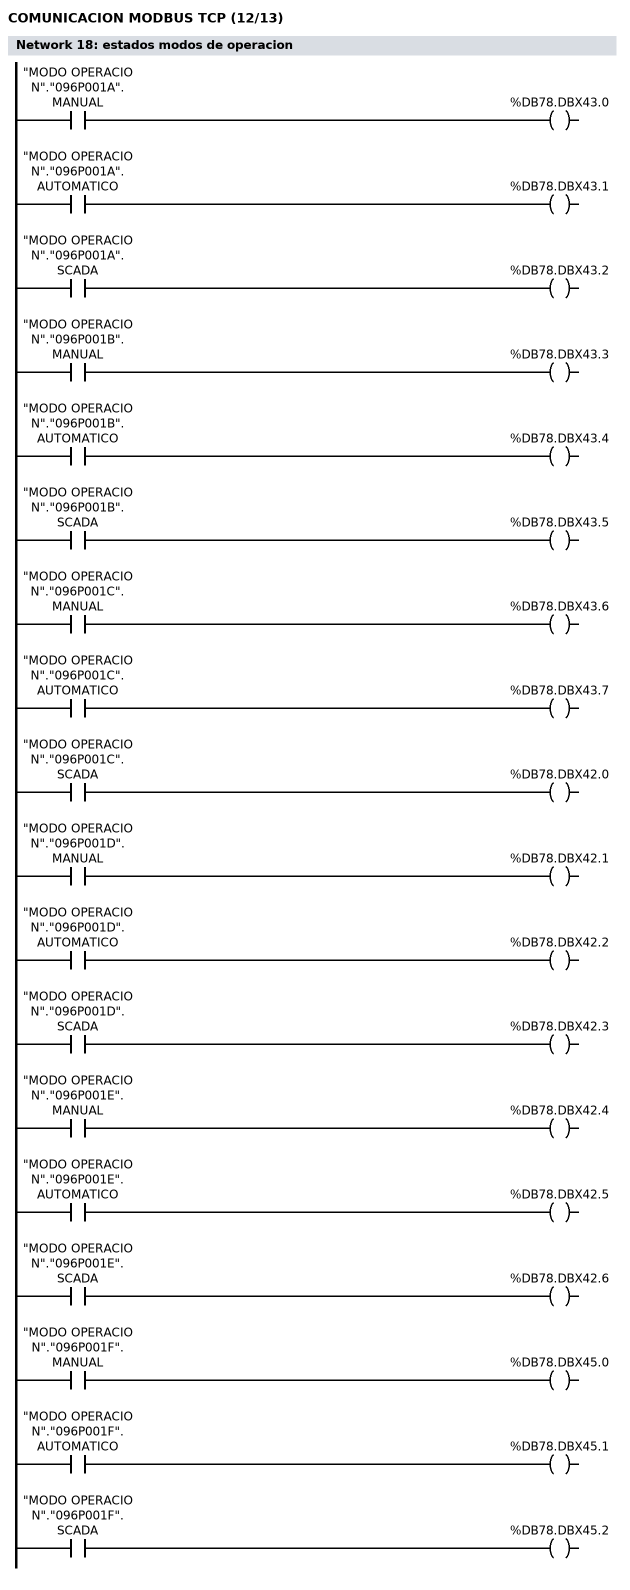
   RUNG wire#powerrail
      Contact( "MODO OPERACION"."096P001A".MANUAL )
      Coil( %DB78.DBX43.0 )
   END_RUNG
   RUNG wire#powerrail
      Contact( "MODO OPERACION"."096P001A".AUTOMATICO )
      Coil( %DB78.DBX43.1 )
   END_RUNG
   RUNG wire#powerrail
      Contact( "MODO OPERACION"."096P001A".SCADA )
      Coil( %DB78.DBX43.2 )
   END_RUNG
   RUNG wire#powerrail
      Contact( "MODO OPERACION"."096P001B".MANUAL )
      Coil( %DB78.DBX43.3 )
   END_RUNG
   RUNG wire#powerrail
      Contact( "MODO OPERACION"."096P001B".AUTOMATICO )
      Coil( %DB78.DBX43.4 )
   END_RUNG
   RUNG wire#powerrail
      Contact( "MODO OPERACION"."096P001B".SCADA )
      Coil( %DB78.DBX43.5 )
   END_RUNG
   RUNG wire#powerrail
      Contact( "MODO OPERACION"."096P001C".MANUAL )
      Coil( %DB78.DBX43.6 )
   END_RUNG
   RUNG wire#powerrail
      Contact( "MODO OPERACION"."096P001C".AUTOMATICO )
      Coil( %DB78.DBX43.7 )
   END_RUNG
   RUNG wire#powerrail
      Contact( "MODO OPERACION"."096P001C".SCADA )
      Coil( %DB78.DBX42.0 )
   END_RUNG
   RUNG wire#powerrail
      Contact( "MODO OPERACION"."096P001D".MANUAL )
      Coil( %DB78.DBX42.1 )
   END_RUNG
   RUNG wire#powerrail
      Contact( "MODO OPERACION"."096P001D".AUTOMATICO )
      Coil( %DB78.DBX42.2 )
   END_RUNG
   RUNG wire#powerrail
      Contact( "MODO OPERACION"."096P001D".SCADA )
      Coil( %DB78.DBX42.3 )
   END_RUNG
   RUNG wire#powerrail
      Contact( "MODO OPERACION"."096P001E".MANUAL )
      Coil( %DB78.DBX42.4 )
   END_RUNG
   RUNG wire#powerrail
      Contact( "MODO OPERACION"."096P001E".AUTOMATICO )
      Coil( %DB78.DBX42.5 )
   END_RUNG
   RUNG wire#powerrail
      Contact( "MODO OPERACION"."096P001E".SCADA )
      Coil( %DB78.DBX42.6 )
   END_RUNG
   RUNG wire#powerrail
      Contact( "MODO OPERACION"."096P001F".MANUAL )
      Coil( %DB78.DBX45.0 )
   END_RUNG
   RUNG wire#powerrail
      Contact( "MODO OPERACION"."096P001F".AUTOMATICO )
      Coil( %DB78.DBX45.1 )
   END_RUNG
   RUNG wire#powerrail
      Contact( "MODO OPERACION"."096P001F".SCADA )
      Coil( %DB78.DBX45.2 )
   END_RUNG
   // the same network as SCL:
   %DB78.DBX43.0 := "MODO OPERACION"."096P001A".MANUAL;
   %DB78.DBX43.1 := "MODO OPERACION"."096P001A".AUTOMATICO;
   %DB78.DBX43.2 := "MODO OPERACION"."096P001A".SCADA;
   %DB78.DBX43.3 := "MODO OPERACION"."096P001B".MANUAL;
   %DB78.DBX43.4 := "MODO OPERACION"."096P001B".AUTOMATICO;
   %DB78.DBX43.5 := "MODO OPERACION"."096P001B".SCADA;
   %DB78.DBX43.6 := "MODO OPERACION"."096P001C".MANUAL;
   %DB78.DBX43.7 := "MODO OPERACION"."096P001C".AUTOMATICO;
   %DB78.DBX42.0 := "MODO OPERACION"."096P001C".SCADA;
   %DB78.DBX42.1 := "MODO OPERACION"."096P001D".MANUAL;
   %DB78.DBX42.2 := "MODO OPERACION"."096P001D".AUTOMATICO;
   %DB78.DBX42.3 := "MODO OPERACION"."096P001D".SCADA;
   %DB78.DBX42.4 := "MODO OPERACION"."096P001E".MANUAL;
   %DB78.DBX42.5 := "MODO OPERACION"."096P001E".AUTOMATICO;
   %DB78.DBX42.6 := "MODO OPERACION"."096P001E".SCADA;
   %DB78.DBX45.0 := "MODO OPERACION"."096P001F".MANUAL;
   %DB78.DBX45.1 := "MODO OPERACION"."096P001F".AUTOMATICO;
   %DB78.DBX45.2 := "MODO OPERACION"."096P001F".SCADA;
END_REGION

REGION Network 19: fallas gnerales
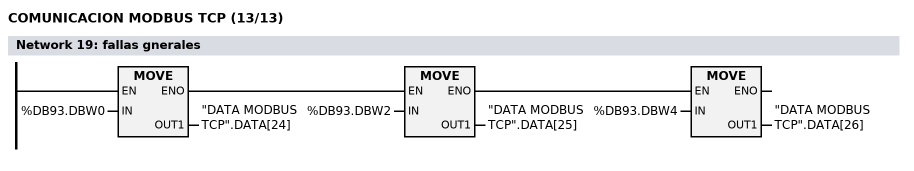
   RUNG wire#powerrail
      Move(in := %DB93.DBW0, out1 => "DATA MODBUS TCP".DATA[24])
      Move(in := %DB93.DBW2, out1 => "DATA MODBUS TCP".DATA[25])
      Move(in := %DB93.DBW4, out1 => "DATA MODBUS TCP".DATA[26])
   END_RUNG
   // the same network as SCL:
   "DATA MODBUS TCP".DATA[24] := %DB93.DBW0;
   "DATA MODBUS TCP".DATA[25] := %DB93.DBW2;
   "DATA MODBUS TCP".DATA[26] := %DB93.DBW4;
END_REGION
END_FUNCTION

FUNCTION "FALLAS" : Void   // FC8, LAD
{ S7_Optimized_Access := 'TRUE' }
VERSION : 0.1
   VAR_TEMP
      "RESET A" : Bool;
      "RESET B" : Bool;
      "RESET C" : Bool;
      "RESET D" : Bool;
      "RESET E" : Bool;
      "RESET F" : Bool;
   END_VAR
BEGIN

REGION Network 1: reset gral
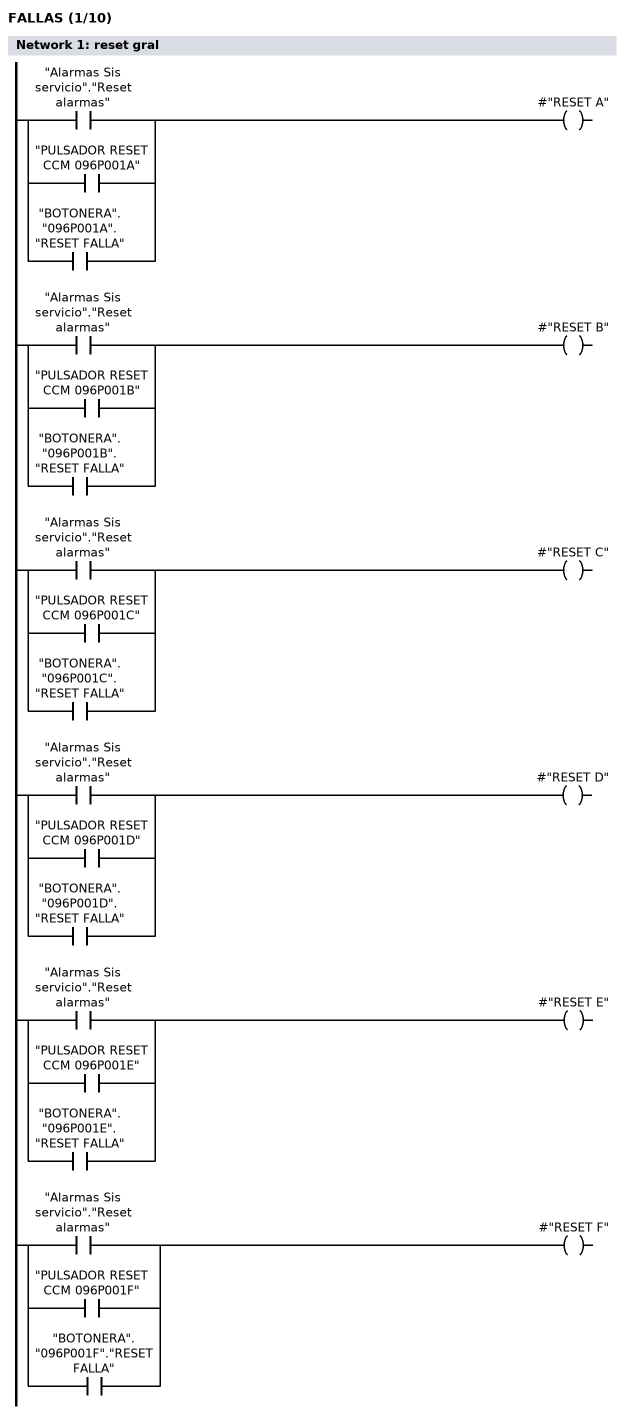
   RUNG wire#powerrail
      Contact( "Alarmas Sis servicio"."Reset alarmas" )
      wire#w1
      Coil( #"RESET A" )
   END_RUNG
   RUNG wire#powerrail
      Contact( "PULSADOR RESET CCM 096P001A" )
   END_RUNG wire#w1
   RUNG wire#powerrail
      Contact( "BOTONERA"."096P001A"."RESET FALLA" )
   END_RUNG wire#w1
   RUNG wire#powerrail
      Contact( "Alarmas Sis servicio"."Reset alarmas" )
      wire#w2
      Coil( #"RESET B" )
   END_RUNG
   RUNG wire#powerrail
      Contact( "PULSADOR RESET CCM 096P001B" )
   END_RUNG wire#w2
   RUNG wire#powerrail
      Contact( "BOTONERA"."096P001B"."RESET FALLA" )
   END_RUNG wire#w2
   RUNG wire#powerrail
      Contact( "Alarmas Sis servicio"."Reset alarmas" )
      wire#w3
      Coil( #"RESET C" )
   END_RUNG
   RUNG wire#powerrail
      Contact( "PULSADOR RESET CCM 096P001C" )
   END_RUNG wire#w3
   RUNG wire#powerrail
      Contact( "BOTONERA"."096P001C"."RESET FALLA" )
   END_RUNG wire#w3
   RUNG wire#powerrail
      Contact( "Alarmas Sis servicio"."Reset alarmas" )
      wire#w4
      Coil( #"RESET D" )
   END_RUNG
   RUNG wire#powerrail
      Contact( "PULSADOR RESET CCM 096P001D" )
   END_RUNG wire#w4
   RUNG wire#powerrail
      Contact( "BOTONERA"."096P001D"."RESET FALLA" )
   END_RUNG wire#w4
   RUNG wire#powerrail
      Contact( "Alarmas Sis servicio"."Reset alarmas" )
      wire#w5
      Coil( #"RESET E" )
   END_RUNG
   RUNG wire#powerrail
      Contact( "PULSADOR RESET CCM 096P001E" )
   END_RUNG wire#w5
   RUNG wire#powerrail
      Contact( "BOTONERA"."096P001E"."RESET FALLA" )
   END_RUNG wire#w5
   RUNG wire#powerrail
      Contact( "Alarmas Sis servicio"."Reset alarmas" )
      wire#w6
      Coil( #"RESET F" )
   END_RUNG
   RUNG wire#powerrail
      Contact( "PULSADOR RESET CCM 096P001F" )
   END_RUNG wire#w6
   RUNG wire#powerrail
      Contact( "BOTONERA"."096P001F"."RESET FALLA" )
   END_RUNG wire#w6
   // the same network as SCL:
   #"RESET A" := "Alarmas Sis servicio"."Reset alarmas" OR "PULSADOR RESET CCM 096P001A" OR "BOTONERA"."096P001A"."RESET FALLA";
   #"RESET B" := "Alarmas Sis servicio"."Reset alarmas" OR "PULSADOR RESET CCM 096P001B" OR "BOTONERA"."096P001B"."RESET FALLA";
   #"RESET C" := "Alarmas Sis servicio"."Reset alarmas" OR "PULSADOR RESET CCM 096P001C" OR "BOTONERA"."096P001C"."RESET FALLA";
   #"RESET D" := "Alarmas Sis servicio"."Reset alarmas" OR "PULSADOR RESET CCM 096P001D" OR "BOTONERA"."096P001D"."RESET FALLA";
   #"RESET E" := "Alarmas Sis servicio"."Reset alarmas" OR "PULSADOR RESET CCM 096P001E" OR "BOTONERA"."096P001E"."RESET FALLA";
   #"RESET F" := "Alarmas Sis servicio"."Reset alarmas" OR "PULSADOR RESET CCM 096P001F" OR "BOTONERA"."096P001F"."RESET FALLA";
END_REGION

REGION Network 2: PARO DE EMERGENCIA GRAL
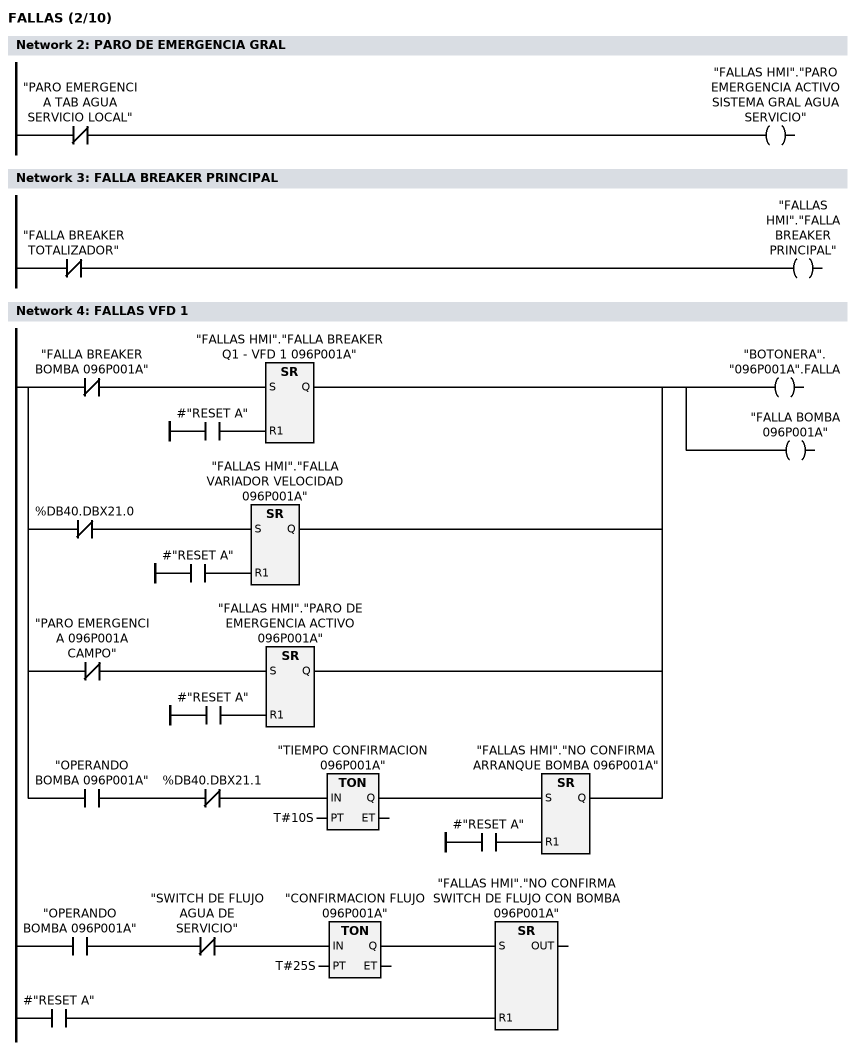
   RUNG wire#powerrail
      I_Contact( "PARO EMERGENCIA TAB AGUA SERVICIO LOCAL" )
      Coil( "FALLAS HMI"."PARO EMERGENCIA ACTIVO SISTEMA GRAL AGUA SERVICIO" )
   END_RUNG
   // the same network as SCL:
   "FALLAS HMI"."PARO EMERGENCIA ACTIVO SISTEMA GRAL AGUA SERVICIO" := NOT "PARO EMERGENCIA TAB AGUA SERVICIO LOCAL";
END_REGION

REGION Network 3: FALLA BREAKER PRINCIPAL
   RUNG wire#powerrail
      I_Contact( "FALLA BREAKER TOTALIZADOR" )
      Coil( "FALLAS HMI"."FALLA BREAKER PRINCIPAL" )
   END_RUNG
   // the same network as SCL:
   "FALLAS HMI"."FALLA BREAKER PRINCIPAL" := NOT "FALLA BREAKER TOTALIZADOR";
END_REGION

REGION Network 4: FALLAS VFD 1
   IF NOT "FALLA BREAKER BOMBA 096P001A" THEN
       "FALLAS HMI"."FALLA BREAKER Q1 - VFD 1 096P001A" := TRUE;   // SR flip-flop
   END_IF;
   IF #"RESET A" THEN "FALLAS HMI"."FALLA BREAKER Q1 - VFD 1 096P001A" := FALSE; END_IF;
   IF NOT %DB40.DBX21.0 THEN
       "FALLAS HMI"."FALLA VARIADOR VELOCIDAD 096P001A" := TRUE;   // SR flip-flop
   END_IF;
   IF #"RESET A" THEN "FALLAS HMI"."FALLA VARIADOR VELOCIDAD 096P001A" := FALSE; END_IF;
   IF NOT "PARO EMERGENCIA 096P001A CAMPO" THEN
       "FALLAS HMI"."PARO DE EMERGENCIA ACTIVO 096P001A" := TRUE;   // SR flip-flop
   END_IF;
   IF #"RESET A" THEN "FALLAS HMI"."PARO DE EMERGENCIA ACTIVO 096P001A" := FALSE; END_IF;
   "TIEMPO CONFIRMACION 096P001A".TON(IN := "OPERANDO BOMBA 096P001A" AND NOT %DB40.DBX21.1, PT := T#10S);
   IF "TIEMPO CONFIRMACION 096P001A".Q THEN
       "FALLAS HMI"."NO CONFIRMA ARRANQUE BOMBA 096P001A" := TRUE;   // SR flip-flop
   END_IF;
   IF #"RESET A" THEN "FALLAS HMI"."NO CONFIRMA ARRANQUE BOMBA 096P001A" := FALSE; END_IF;
   "BOTONERA"."096P001A".FALLA := "FALLAS HMI"."FALLA BREAKER Q1 - VFD 1 096P001A" OR "FALLAS HMI"."FALLA VARIADOR VELOCIDAD 096P001A" OR "FALLAS HMI"."PARO DE EMERGENCIA ACTIVO 096P001A" OR "FALLAS HMI"."NO CONFIRMA ARRANQUE BOMBA 096P001A";
   "FALLA BOMBA 096P001A" := "BOTONERA"."096P001A".FALLA;
   "CONFIRMACION FLUJO 096P001A".TON(IN := "OPERANDO BOMBA 096P001A" AND NOT "SWITCH DE FLUJO AGUA DE SERVICIO",
                           PT := T#25S);
   IF "CONFIRMACION FLUJO 096P001A".Q THEN
       "FALLAS HMI"."NO CONFIRMA SWITCH DE FLUJO CON BOMBA 096P001A" := TRUE;   // SR flip-flop
   END_IF;
   IF #"RESET A" THEN "FALLAS HMI"."NO CONFIRMA SWITCH DE FLUJO CON BOMBA 096P001A" := FALSE; END_IF;
END_REGION

REGION Network 5: FALLAS VFD 2
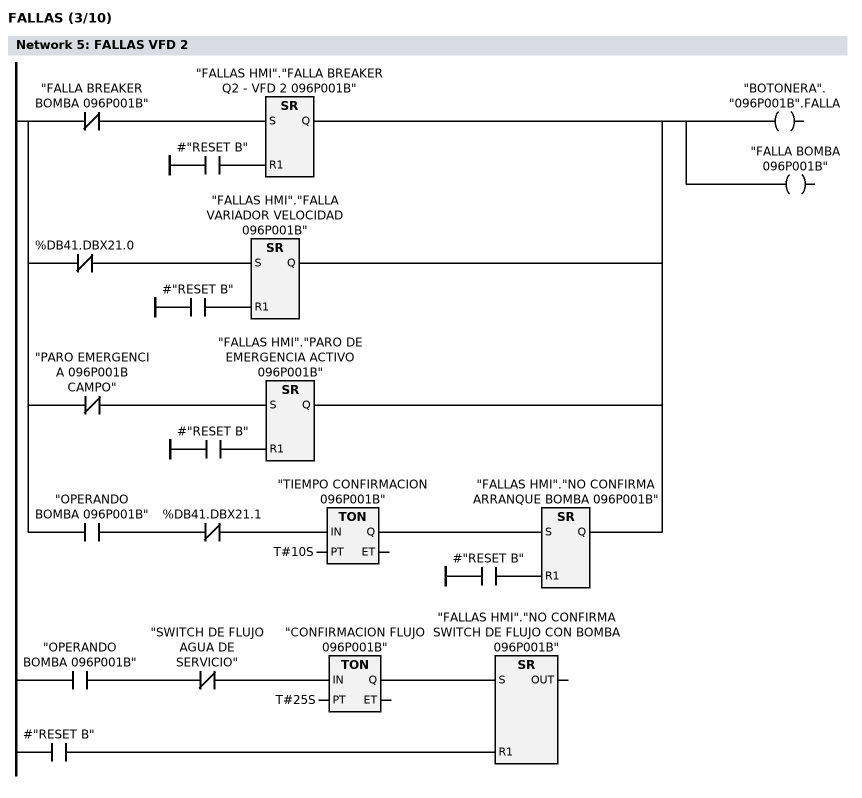
   IF NOT "FALLA BREAKER BOMBA 096P001B" THEN
       "FALLAS HMI"."FALLA BREAKER Q2 - VFD 2 096P001B" := TRUE;   // SR flip-flop
   END_IF;
   IF #"RESET B" THEN "FALLAS HMI"."FALLA BREAKER Q2 - VFD 2 096P001B" := FALSE; END_IF;
   IF NOT %DB41.DBX21.0 THEN
       "FALLAS HMI"."FALLA VARIADOR VELOCIDAD 096P001B" := TRUE;   // SR flip-flop
   END_IF;
   IF #"RESET B" THEN "FALLAS HMI"."FALLA VARIADOR VELOCIDAD 096P001B" := FALSE; END_IF;
   IF NOT "PARO EMERGENCIA 096P001B CAMPO" THEN
       "FALLAS HMI"."PARO DE EMERGENCIA ACTIVO 096P001B" := TRUE;   // SR flip-flop
   END_IF;
   IF #"RESET B" THEN "FALLAS HMI"."PARO DE EMERGENCIA ACTIVO 096P001B" := FALSE; END_IF;
   "TIEMPO CONFIRMACION 096P001B".TON(IN := "OPERANDO BOMBA 096P001B" AND NOT %DB41.DBX21.1, PT := T#10S);
   IF "TIEMPO CONFIRMACION 096P001B".Q THEN
       "FALLAS HMI"."NO CONFIRMA ARRANQUE BOMBA 096P001B" := TRUE;   // SR flip-flop
   END_IF;
   IF #"RESET B" THEN "FALLAS HMI"."NO CONFIRMA ARRANQUE BOMBA 096P001B" := FALSE; END_IF;
   "BOTONERA"."096P001B".FALLA := "FALLAS HMI"."FALLA BREAKER Q2 - VFD 2 096P001B" OR "FALLAS HMI"."FALLA VARIADOR VELOCIDAD 096P001B" OR "FALLAS HMI"."PARO DE EMERGENCIA ACTIVO 096P001B" OR "FALLAS HMI"."NO CONFIRMA ARRANQUE BOMBA 096P001B";
   "FALLA BOMBA 096P001B" := "BOTONERA"."096P001B".FALLA;
   "CONFIRMACION FLUJO 096P001B".TON(IN := "OPERANDO BOMBA 096P001B" AND NOT "SWITCH DE FLUJO AGUA DE SERVICIO",
                           PT := T#25S);
   IF "CONFIRMACION FLUJO 096P001B".Q THEN
       "FALLAS HMI"."NO CONFIRMA SWITCH DE FLUJO CON BOMBA 096P001B" := TRUE;   // SR flip-flop
   END_IF;
   IF #"RESET B" THEN "FALLAS HMI"."NO CONFIRMA SWITCH DE FLUJO CON BOMBA 096P001B" := FALSE; END_IF;
END_REGION

REGION Network 6: FALLAS VFD 3
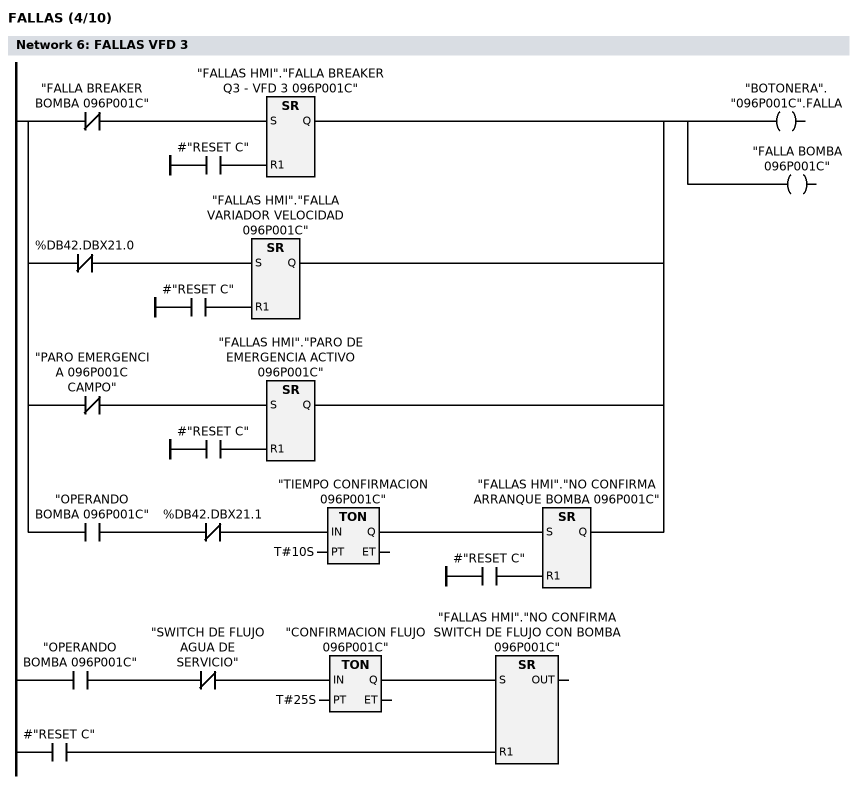
   IF NOT "FALLA BREAKER BOMBA 096P001C" THEN
       "FALLAS HMI"."FALLA BREAKER Q3 - VFD 3 096P001C" := TRUE;   // SR flip-flop
   END_IF;
   IF #"RESET C" THEN "FALLAS HMI"."FALLA BREAKER Q3 - VFD 3 096P001C" := FALSE; END_IF;
   IF NOT %DB42.DBX21.0 THEN
       "FALLAS HMI"."FALLA VARIADOR VELOCIDAD 096P001C" := TRUE;   // SR flip-flop
   END_IF;
   IF #"RESET C" THEN "FALLAS HMI"."FALLA VARIADOR VELOCIDAD 096P001C" := FALSE; END_IF;
   IF NOT "PARO EMERGENCIA 096P001C CAMPO" THEN
       "FALLAS HMI"."PARO DE EMERGENCIA ACTIVO 096P001C" := TRUE;   // SR flip-flop
   END_IF;
   IF #"RESET C" THEN "FALLAS HMI"."PARO DE EMERGENCIA ACTIVO 096P001C" := FALSE; END_IF;
   "TIEMPO CONFIRMACION 096P001C".TON(IN := "OPERANDO BOMBA 096P001C" AND NOT %DB42.DBX21.1, PT := T#10S);
   IF "TIEMPO CONFIRMACION 096P001C".Q THEN
       "FALLAS HMI"."NO CONFIRMA ARRANQUE BOMBA 096P001C" := TRUE;   // SR flip-flop
   END_IF;
   IF #"RESET C" THEN "FALLAS HMI"."NO CONFIRMA ARRANQUE BOMBA 096P001C" := FALSE; END_IF;
   "BOTONERA"."096P001C".FALLA := "FALLAS HMI"."FALLA BREAKER Q3 - VFD 3 096P001C" OR "FALLAS HMI"."FALLA VARIADOR VELOCIDAD 096P001C" OR "FALLAS HMI"."PARO DE EMERGENCIA ACTIVO 096P001C" OR "FALLAS HMI"."NO CONFIRMA ARRANQUE BOMBA 096P001C";
   "FALLA BOMBA 096P001C" := "BOTONERA"."096P001C".FALLA;
   "CONFIRMACION FLUJO 096P001C".TON(IN := "OPERANDO BOMBA 096P001C" AND NOT "SWITCH DE FLUJO AGUA DE SERVICIO",
                           PT := T#25S);
   IF "CONFIRMACION FLUJO 096P001C".Q THEN
       "FALLAS HMI"."NO CONFIRMA SWITCH DE FLUJO CON BOMBA 096P001C" := TRUE;   // SR flip-flop
   END_IF;
   IF #"RESET C" THEN "FALLAS HMI"."NO CONFIRMA SWITCH DE FLUJO CON BOMBA 096P001C" := FALSE; END_IF;
END_REGION

REGION Network 7: FALLAS VFD 4
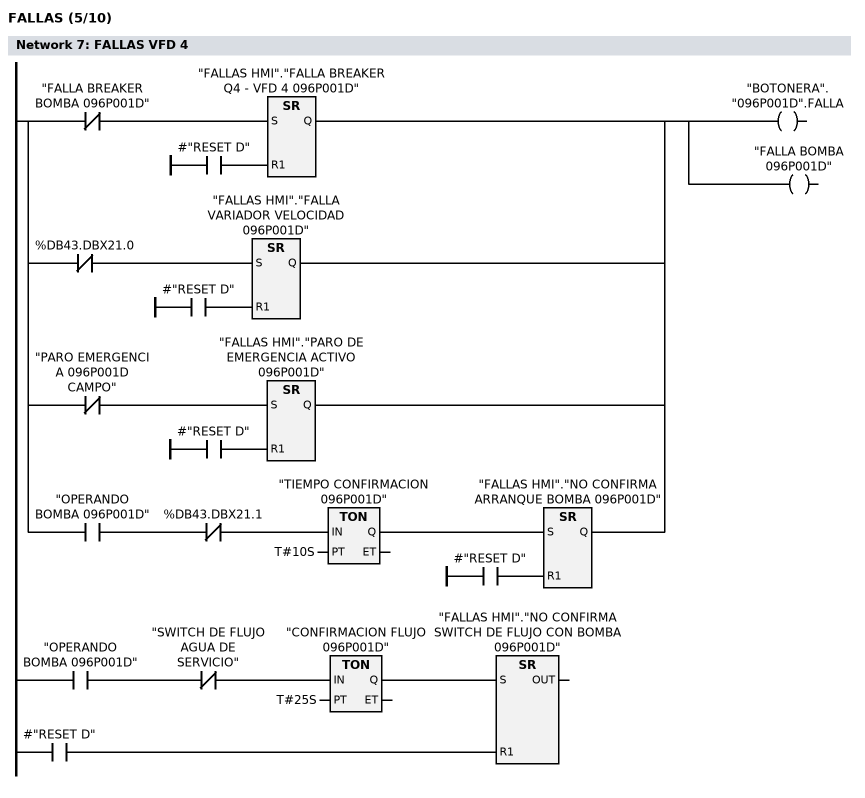
   IF NOT "FALLA BREAKER BOMBA 096P001D" THEN
       "FALLAS HMI"."FALLA BREAKER Q4 - VFD 4 096P001D" := TRUE;   // SR flip-flop
   END_IF;
   IF #"RESET D" THEN "FALLAS HMI"."FALLA BREAKER Q4 - VFD 4 096P001D" := FALSE; END_IF;
   IF NOT %DB43.DBX21.0 THEN
       "FALLAS HMI"."FALLA VARIADOR VELOCIDAD 096P001D" := TRUE;   // SR flip-flop
   END_IF;
   IF #"RESET D" THEN "FALLAS HMI"."FALLA VARIADOR VELOCIDAD 096P001D" := FALSE; END_IF;
   IF NOT "PARO EMERGENCIA 096P001D CAMPO" THEN
       "FALLAS HMI"."PARO DE EMERGENCIA ACTIVO 096P001D" := TRUE;   // SR flip-flop
   END_IF;
   IF #"RESET D" THEN "FALLAS HMI"."PARO DE EMERGENCIA ACTIVO 096P001D" := FALSE; END_IF;
   "TIEMPO CONFIRMACION 096P001D".TON(IN := "OPERANDO BOMBA 096P001D" AND NOT %DB43.DBX21.1, PT := T#10S);
   IF "TIEMPO CONFIRMACION 096P001D".Q THEN
       "FALLAS HMI"."NO CONFIRMA ARRANQUE BOMBA 096P001D" := TRUE;   // SR flip-flop
   END_IF;
   IF #"RESET D" THEN "FALLAS HMI"."NO CONFIRMA ARRANQUE BOMBA 096P001D" := FALSE; END_IF;
   "BOTONERA"."096P001D".FALLA := "FALLAS HMI"."FALLA BREAKER Q4 - VFD 4 096P001D" OR "FALLAS HMI"."FALLA VARIADOR VELOCIDAD 096P001D" OR "FALLAS HMI"."PARO DE EMERGENCIA ACTIVO 096P001D" OR "FALLAS HMI"."NO CONFIRMA ARRANQUE BOMBA 096P001D";
   "FALLA BOMBA 096P001D" := "BOTONERA"."096P001D".FALLA;
   "CONFIRMACION FLUJO 096P001D".TON(IN := "OPERANDO BOMBA 096P001D" AND NOT "SWITCH DE FLUJO AGUA DE SERVICIO",
                           PT := T#25S);
   IF "CONFIRMACION FLUJO 096P001D".Q THEN
       "FALLAS HMI"."NO CONFIRMA SWITCH DE FLUJO CON BOMBA 096P001D" := TRUE;   // SR flip-flop
   END_IF;
   IF #"RESET D" THEN "FALLAS HMI"."NO CONFIRMA SWITCH DE FLUJO CON BOMBA 096P001D" := FALSE; END_IF;
END_REGION

REGION Network 8: FALLAS VFD 5
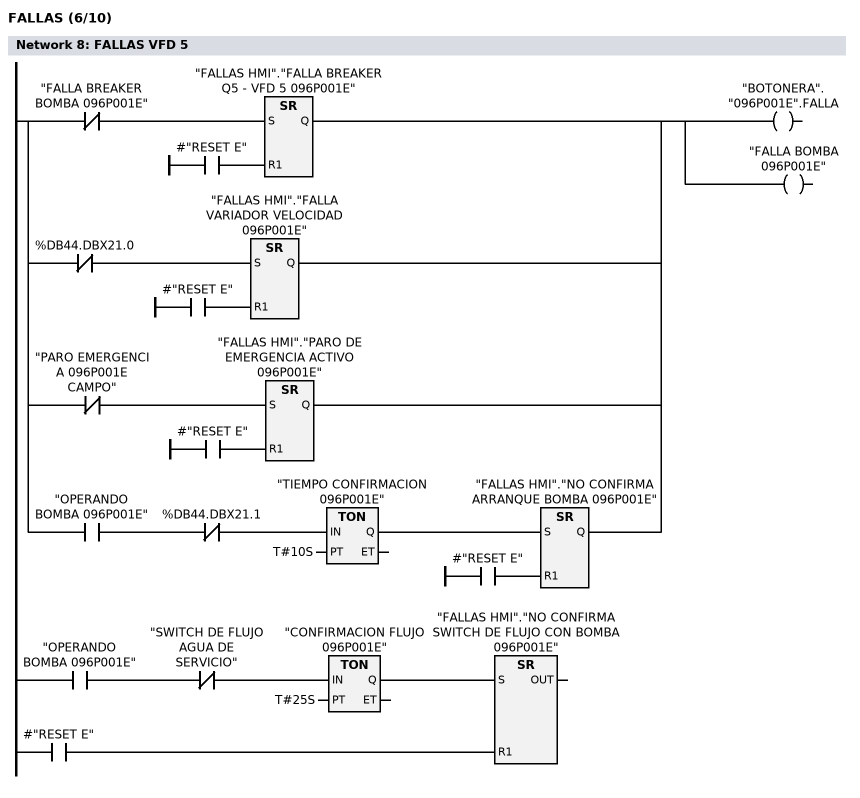
   IF NOT "FALLA BREAKER BOMBA 096P001E" THEN
       "FALLAS HMI"."FALLA BREAKER Q5 - VFD 5 096P001E" := TRUE;   // SR flip-flop
   END_IF;
   IF #"RESET E" THEN "FALLAS HMI"."FALLA BREAKER Q5 - VFD 5 096P001E" := FALSE; END_IF;
   IF NOT %DB44.DBX21.0 THEN
       "FALLAS HMI"."FALLA VARIADOR VELOCIDAD 096P001E" := TRUE;   // SR flip-flop
   END_IF;
   IF #"RESET E" THEN "FALLAS HMI"."FALLA VARIADOR VELOCIDAD 096P001E" := FALSE; END_IF;
   IF NOT "PARO EMERGENCIA 096P001E CAMPO" THEN
       "FALLAS HMI"."PARO DE EMERGENCIA ACTIVO 096P001E" := TRUE;   // SR flip-flop
   END_IF;
   IF #"RESET E" THEN "FALLAS HMI"."PARO DE EMERGENCIA ACTIVO 096P001E" := FALSE; END_IF;
   "TIEMPO CONFIRMACION 096P001E".TON(IN := "OPERANDO BOMBA 096P001E" AND NOT %DB44.DBX21.1, PT := T#10S);
   IF "TIEMPO CONFIRMACION 096P001E".Q THEN
       "FALLAS HMI"."NO CONFIRMA ARRANQUE BOMBA 096P001E" := TRUE;   // SR flip-flop
   END_IF;
   IF #"RESET E" THEN "FALLAS HMI"."NO CONFIRMA ARRANQUE BOMBA 096P001E" := FALSE; END_IF;
   "BOTONERA"."096P001E".FALLA := "FALLAS HMI"."FALLA BREAKER Q5 - VFD 5 096P001E" OR "FALLAS HMI"."FALLA VARIADOR VELOCIDAD 096P001E" OR "FALLAS HMI"."PARO DE EMERGENCIA ACTIVO 096P001E" OR "FALLAS HMI"."NO CONFIRMA ARRANQUE BOMBA 096P001E";
   "FALLA BOMBA 096P001E" := "BOTONERA"."096P001E".FALLA;
   "CONFIRMACION FLUJO 096P001E".TON(IN := "OPERANDO BOMBA 096P001E" AND NOT "SWITCH DE FLUJO AGUA DE SERVICIO",
                           PT := T#25S);
   IF "CONFIRMACION FLUJO 096P001E".Q THEN
       "FALLAS HMI"."NO CONFIRMA SWITCH DE FLUJO CON BOMBA 096P001E" := TRUE;   // SR flip-flop
   END_IF;
   IF #"RESET E" THEN "FALLAS HMI"."NO CONFIRMA SWITCH DE FLUJO CON BOMBA 096P001E" := FALSE; END_IF;
END_REGION

REGION Network 9: FALLAS VFD 6
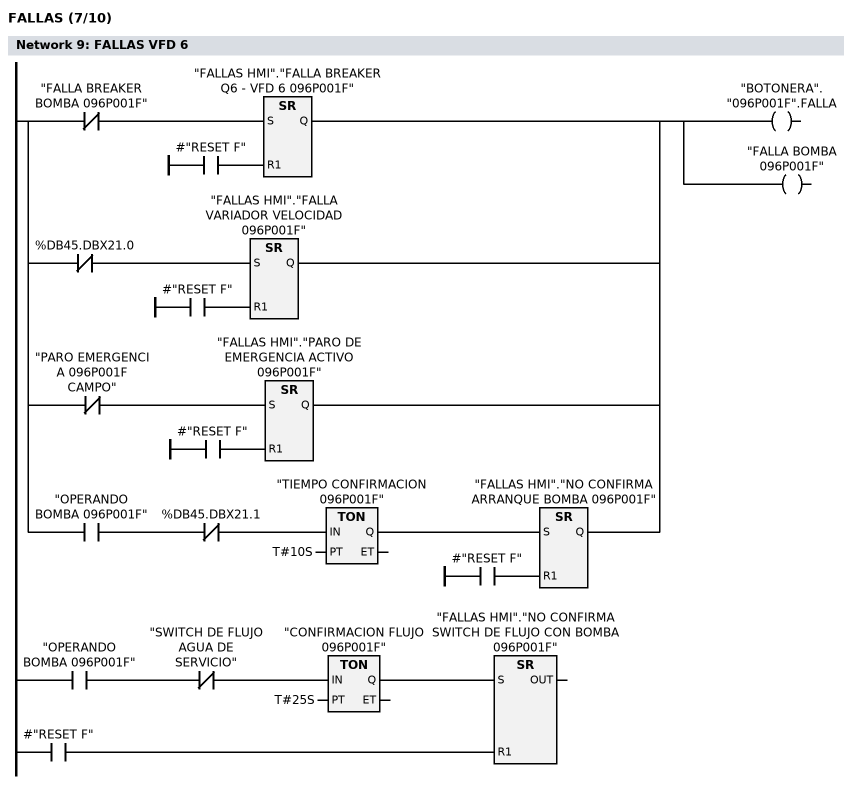
   IF NOT "FALLA BREAKER BOMBA 096P001F" THEN
       "FALLAS HMI"."FALLA BREAKER Q6 - VFD 6 096P001F" := TRUE;   // SR flip-flop
   END_IF;
   IF #"RESET F" THEN "FALLAS HMI"."FALLA BREAKER Q6 - VFD 6 096P001F" := FALSE; END_IF;
   IF NOT %DB45.DBX21.0 THEN
       "FALLAS HMI"."FALLA VARIADOR VELOCIDAD 096P001F" := TRUE;   // SR flip-flop
   END_IF;
   IF #"RESET F" THEN "FALLAS HMI"."FALLA VARIADOR VELOCIDAD 096P001F" := FALSE; END_IF;
   IF NOT "PARO EMERGENCIA 096P001F CAMPO" THEN
       "FALLAS HMI"."PARO DE EMERGENCIA ACTIVO 096P001F" := TRUE;   // SR flip-flop
   END_IF;
   IF #"RESET F" THEN "FALLAS HMI"."PARO DE EMERGENCIA ACTIVO 096P001F" := FALSE; END_IF;
   "TIEMPO CONFIRMACION 096P001F".TON(IN := "OPERANDO BOMBA 096P001F" AND NOT %DB45.DBX21.1, PT := T#10S);
   IF "TIEMPO CONFIRMACION 096P001F".Q THEN
       "FALLAS HMI"."NO CONFIRMA ARRANQUE BOMBA 096P001F" := TRUE;   // SR flip-flop
   END_IF;
   IF #"RESET F" THEN "FALLAS HMI"."NO CONFIRMA ARRANQUE BOMBA 096P001F" := FALSE; END_IF;
   "BOTONERA"."096P001F".FALLA := "FALLAS HMI"."FALLA BREAKER Q6 - VFD 6 096P001F" OR "FALLAS HMI"."FALLA VARIADOR VELOCIDAD 096P001F" OR "FALLAS HMI"."PARO DE EMERGENCIA ACTIVO 096P001F" OR "FALLAS HMI"."NO CONFIRMA ARRANQUE BOMBA 096P001F";
   "FALLA BOMBA 096P001F" := "BOTONERA"."096P001F".FALLA;
   "CONFIRMACION FLUJO 096P001F".TON(IN := "OPERANDO BOMBA 096P001F" AND NOT "SWITCH DE FLUJO AGUA DE SERVICIO",
                           PT := T#25S);
   IF "CONFIRMACION FLUJO 096P001F".Q THEN
       "FALLAS HMI"."NO CONFIRMA SWITCH DE FLUJO CON BOMBA 096P001F" := TRUE;   // SR flip-flop
   END_IF;
   IF #"RESET F" THEN "FALLAS HMI"."NO CONFIRMA SWITCH DE FLUJO CON BOMBA 096P001F" := FALSE; END_IF;
END_REGION

REGION Network 10: FALLA BAJA PRESION EN SUCCION
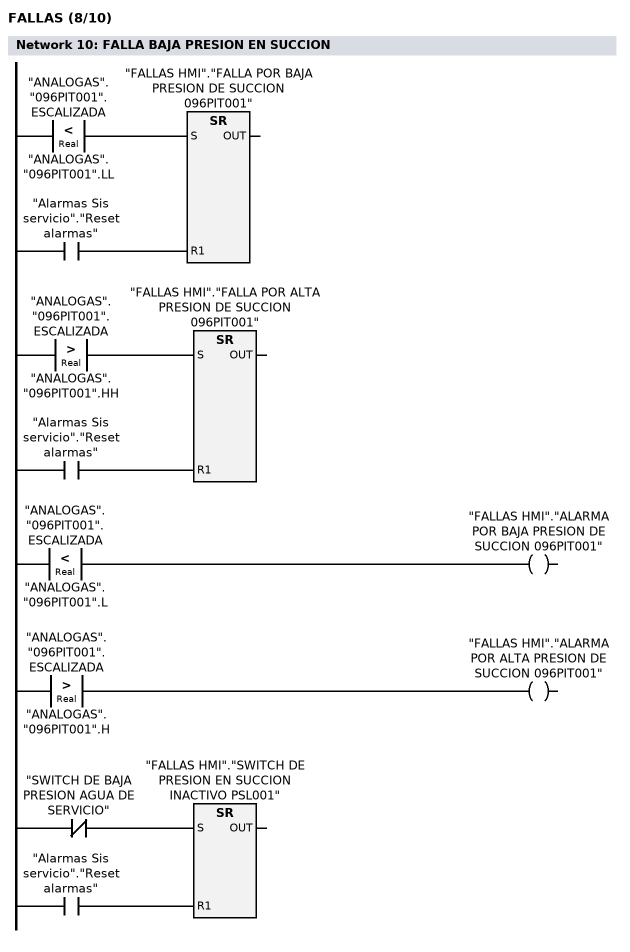
   RUNG wire#powerrail
      { S7_Templates := "SrcType := Real" } LT_Contact(in1 := "ANALOGAS"."096PIT001".ESCALIZADA, in2 := "ANALOGAS"."096PIT001".LL)
      S_SR(operand := "FALLAS HMI"."FALLA POR BAJA PRESION DE SUCCION 096PIT001", r1 := wire#w1)
   END_RUNG
   RUNG wire#powerrail
      Contact( "Alarmas Sis servicio"."Reset alarmas" )
   END_RUNG wire#w1
   RUNG wire#powerrail
      { S7_Templates := "SrcType := Real" } GT_Contact(in1 := "ANALOGAS"."096PIT001".ESCALIZADA, in2 := "ANALOGAS"."096PIT001".HH)
      S_SR(operand := "FALLAS HMI"."FALLA POR ALTA PRESION DE SUCCION 096PIT001", r1 := wire#w2)
   END_RUNG
   RUNG wire#powerrail
      Contact( "Alarmas Sis servicio"."Reset alarmas" )
   END_RUNG wire#w2
   RUNG wire#powerrail
      { S7_Templates := "SrcType := Real" } LT_Contact(in1 := "ANALOGAS"."096PIT001".ESCALIZADA, in2 := "ANALOGAS"."096PIT001".L)
      Coil( "FALLAS HMI"."ALARMA POR BAJA PRESION DE SUCCION 096PIT001" )
   END_RUNG
   RUNG wire#powerrail
      { S7_Templates := "SrcType := Real" } GT_Contact(in1 := "ANALOGAS"."096PIT001".ESCALIZADA, in2 := "ANALOGAS"."096PIT001".H)
      Coil( "FALLAS HMI"."ALARMA POR ALTA PRESION DE SUCCION 096PIT001" )
   END_RUNG
   RUNG wire#powerrail
      I_Contact( "SWITCH DE BAJA PRESION AGUA DE SERVICIO" )
      S_SR(operand := "FALLAS HMI"."SWITCH DE PRESION EN SUCCION INACTIVO PSL001", r1 := wire#w3)
   END_RUNG
   RUNG wire#powerrail
      Contact( "Alarmas Sis servicio"."Reset alarmas" )
   END_RUNG wire#w3
   // the same network as SCL:
   IF "ANALOGAS"."096PIT001".ESCALIZADA < "ANALOGAS"."096PIT001".LL THEN
       "FALLAS HMI"."FALLA POR BAJA PRESION DE SUCCION 096PIT001" := TRUE;   // SR flip-flop
   END_IF;
   IF "Alarmas Sis servicio"."Reset alarmas" THEN
       "FALLAS HMI"."FALLA POR BAJA PRESION DE SUCCION 096PIT001" := FALSE;
   END_IF;
   IF "ANALOGAS"."096PIT001".ESCALIZADA > "ANALOGAS"."096PIT001".HH THEN
       "FALLAS HMI"."FALLA POR ALTA PRESION DE SUCCION 096PIT001" := TRUE;   // SR flip-flop
   END_IF;
   IF "Alarmas Sis servicio"."Reset alarmas" THEN
       "FALLAS HMI"."FALLA POR ALTA PRESION DE SUCCION 096PIT001" := FALSE;
   END_IF;
   "FALLAS HMI"."ALARMA POR BAJA PRESION DE SUCCION 096PIT001" := "ANALOGAS"."096PIT001".ESCALIZADA < "ANALOGAS"."096PIT001".L;
   "FALLAS HMI"."ALARMA POR ALTA PRESION DE SUCCION 096PIT001" := "ANALOGAS"."096PIT001".ESCALIZADA > "ANALOGAS"."096PIT001".H;
   IF NOT "SWITCH DE BAJA PRESION AGUA DE SERVICIO" THEN
       "FALLAS HMI"."SWITCH DE PRESION EN SUCCION INACTIVO PSL001" := TRUE;   // SR flip-flop
   END_IF;
   IF "Alarmas Sis servicio"."Reset alarmas" THEN
       "FALLAS HMI"."SWITCH DE PRESION EN SUCCION INACTIVO PSL001" := FALSE;
   END_IF;
END_REGION

REGION Network 11: FALLA BAJA PRESION EN DESCARGA
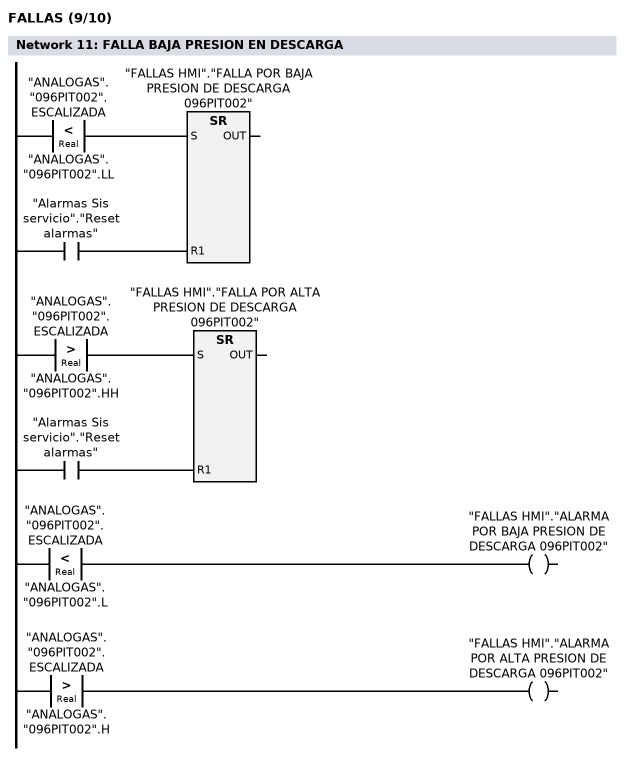
   RUNG wire#powerrail
      { S7_Templates := "SrcType := Real" } LT_Contact(in1 := "ANALOGAS"."096PIT002".ESCALIZADA, in2 := "ANALOGAS"."096PIT002".LL)
      S_SR(operand := "FALLAS HMI"."FALLA POR BAJA PRESION DE DESCARGA 096PIT002", r1 := wire#w1)
   END_RUNG
   RUNG wire#powerrail
      Contact( "Alarmas Sis servicio"."Reset alarmas" )
   END_RUNG wire#w1
   RUNG wire#powerrail
      { S7_Templates := "SrcType := Real" } GT_Contact(in1 := "ANALOGAS"."096PIT002".ESCALIZADA, in2 := "ANALOGAS"."096PIT002".HH)
      S_SR(operand := "FALLAS HMI"."FALLA POR ALTA PRESION DE DESCARGA 096PIT002", r1 := wire#w2)
   END_RUNG
   RUNG wire#powerrail
      Contact( "Alarmas Sis servicio"."Reset alarmas" )
   END_RUNG wire#w2
   RUNG wire#powerrail
      { S7_Templates := "SrcType := Real" } LT_Contact(in1 := "ANALOGAS"."096PIT002".ESCALIZADA, in2 := "ANALOGAS"."096PIT002".L)
      Coil( "FALLAS HMI"."ALARMA POR BAJA PRESION DE DESCARGA 096PIT002" )
   END_RUNG
   RUNG wire#powerrail
      { S7_Templates := "SrcType := Real" } GT_Contact(in1 := "ANALOGAS"."096PIT002".ESCALIZADA, in2 := "ANALOGAS"."096PIT002".H)
      Coil( "FALLAS HMI"."ALARMA POR ALTA PRESION DE DESCARGA 096PIT002" )
   END_RUNG
   // the same network as SCL:
   IF "ANALOGAS"."096PIT002".ESCALIZADA < "ANALOGAS"."096PIT002".LL THEN
       "FALLAS HMI"."FALLA POR BAJA PRESION DE DESCARGA 096PIT002" := TRUE;   // SR flip-flop
   END_IF;
   IF "Alarmas Sis servicio"."Reset alarmas" THEN
       "FALLAS HMI"."FALLA POR BAJA PRESION DE DESCARGA 096PIT002" := FALSE;
   END_IF;
   IF "ANALOGAS"."096PIT002".ESCALIZADA > "ANALOGAS"."096PIT002".HH THEN
       "FALLAS HMI"."FALLA POR ALTA PRESION DE DESCARGA 096PIT002" := TRUE;   // SR flip-flop
   END_IF;
   IF "Alarmas Sis servicio"."Reset alarmas" THEN
       "FALLAS HMI"."FALLA POR ALTA PRESION DE DESCARGA 096PIT002" := FALSE;
   END_IF;
   "FALLAS HMI"."ALARMA POR BAJA PRESION DE DESCARGA 096PIT002" := "ANALOGAS"."096PIT002".ESCALIZADA < "ANALOGAS"."096PIT002".L;
   "FALLAS HMI"."ALARMA POR ALTA PRESION DE DESCARGA 096PIT002" := "ANALOGAS"."096PIT002".ESCALIZADA > "ANALOGAS"."096PIT002".H;
END_REGION

REGION Network 12: FALLAS GRAL
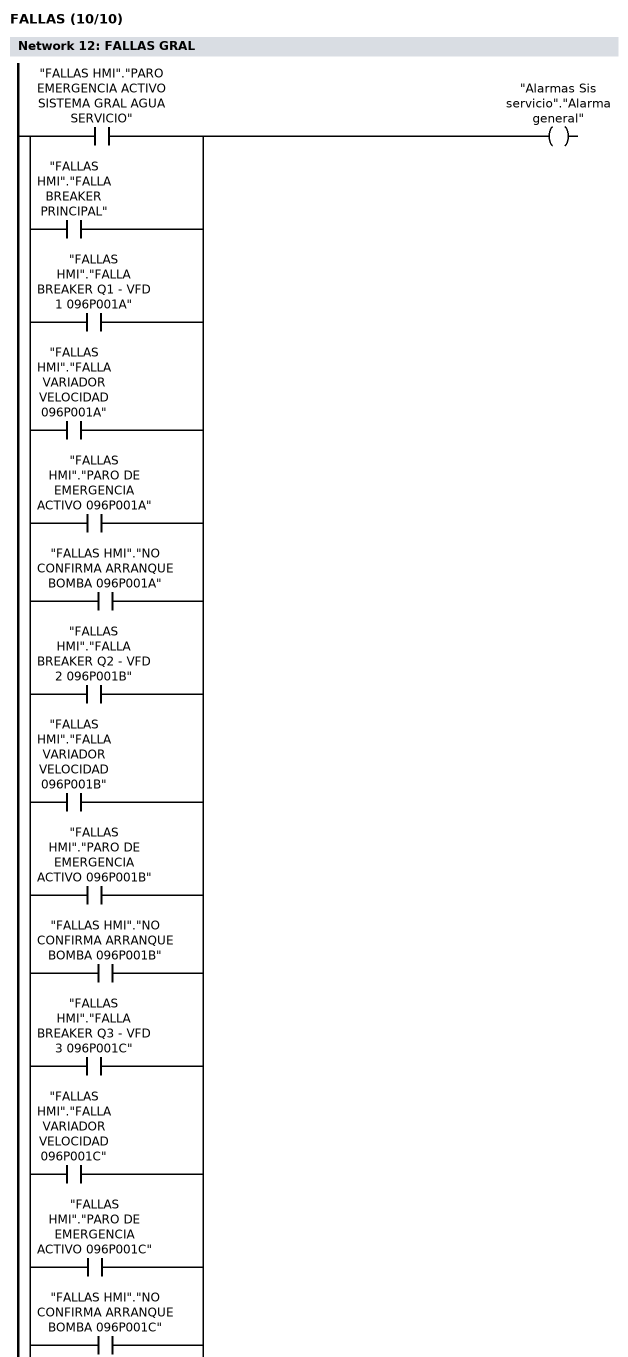
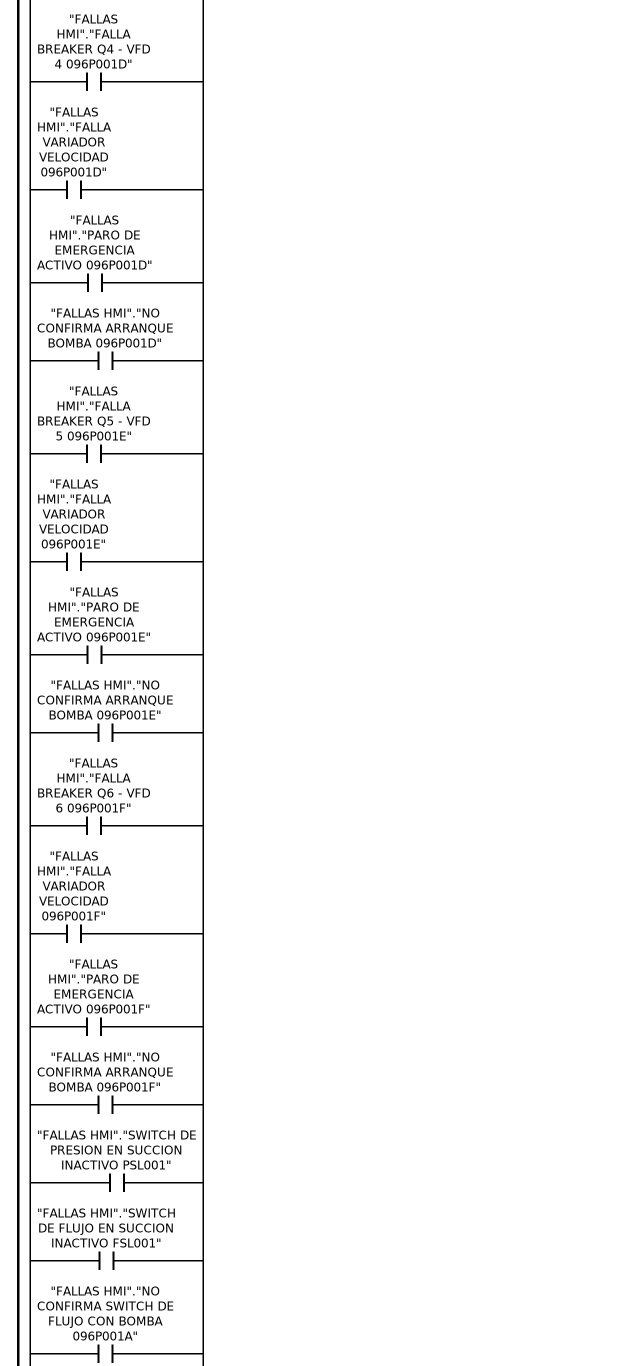
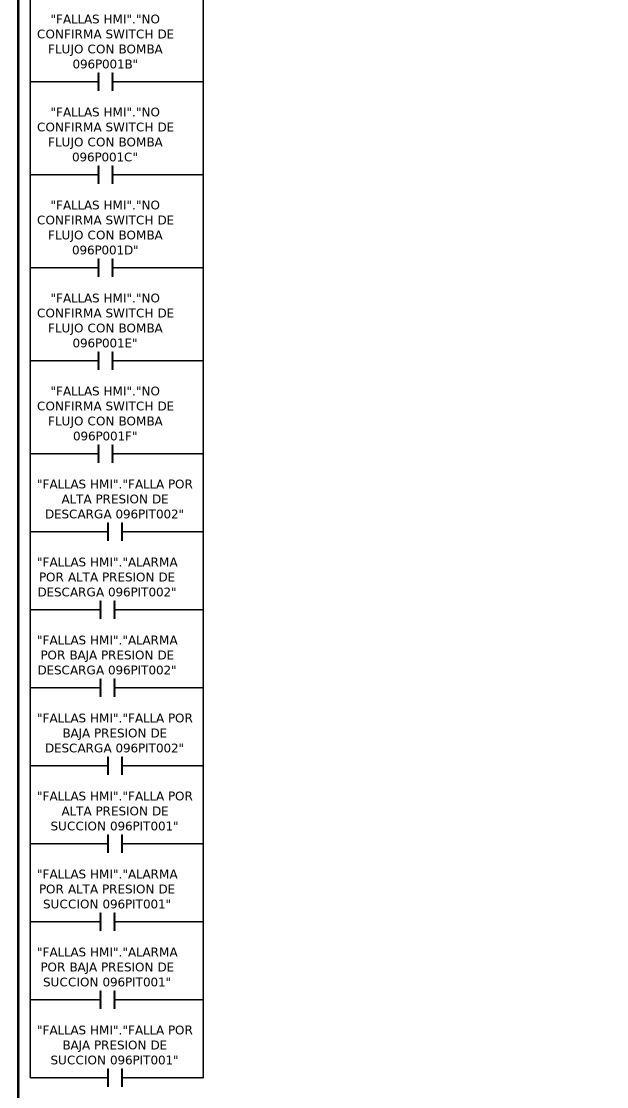
   RUNG wire#powerrail
      Contact( "FALLAS HMI"."PARO EMERGENCIA ACTIVO SISTEMA GRAL AGUA SERVICIO" )
      wire#w1
      Coil( "Alarmas Sis servicio"."Alarma general" )
   END_RUNG
   RUNG wire#powerrail
      Contact( "FALLAS HMI"."FALLA BREAKER PRINCIPAL" )
   END_RUNG wire#w1
   RUNG wire#powerrail
      Contact( "FALLAS HMI"."FALLA BREAKER Q1 - VFD 1 096P001A" )
   END_RUNG wire#w1
   RUNG wire#powerrail
      Contact( "FALLAS HMI"."FALLA VARIADOR VELOCIDAD 096P001A" )
   END_RUNG wire#w1
   RUNG wire#powerrail
      Contact( "FALLAS HMI"."PARO DE EMERGENCIA ACTIVO 096P001A" )
   END_RUNG wire#w1
   RUNG wire#powerrail
      Contact( "FALLAS HMI"."NO CONFIRMA ARRANQUE BOMBA 096P001A" )
   END_RUNG wire#w1
   RUNG wire#powerrail
      Contact( "FALLAS HMI"."FALLA BREAKER Q2 - VFD 2 096P001B" )
   END_RUNG wire#w1
   RUNG wire#powerrail
      Contact( "FALLAS HMI"."FALLA VARIADOR VELOCIDAD 096P001B" )
   END_RUNG wire#w1
   RUNG wire#powerrail
      Contact( "FALLAS HMI"."PARO DE EMERGENCIA ACTIVO 096P001B" )
   END_RUNG wire#w1
   RUNG wire#powerrail
      Contact( "FALLAS HMI"."NO CONFIRMA ARRANQUE BOMBA 096P001B" )
   END_RUNG wire#w1
   RUNG wire#powerrail
      Contact( "FALLAS HMI"."FALLA BREAKER Q3 - VFD 3 096P001C" )
   END_RUNG wire#w1
   RUNG wire#powerrail
      Contact( "FALLAS HMI"."FALLA VARIADOR VELOCIDAD 096P001C" )
   END_RUNG wire#w1
   RUNG wire#powerrail
      Contact( "FALLAS HMI"."PARO DE EMERGENCIA ACTIVO 096P001C" )
   END_RUNG wire#w1
   RUNG wire#powerrail
      Contact( "FALLAS HMI"."NO CONFIRMA ARRANQUE BOMBA 096P001C" )
   END_RUNG wire#w1
   RUNG wire#powerrail
      Contact( "FALLAS HMI"."FALLA BREAKER Q4 - VFD 4 096P001D" )
   END_RUNG wire#w1
   RUNG wire#powerrail
      Contact( "FALLAS HMI"."FALLA VARIADOR VELOCIDAD 096P001D" )
   END_RUNG wire#w1
   RUNG wire#powerrail
      Contact( "FALLAS HMI"."PARO DE EMERGENCIA ACTIVO 096P001D" )
   END_RUNG wire#w1
   RUNG wire#powerrail
      Contact( "FALLAS HMI"."NO CONFIRMA ARRANQUE BOMBA 096P001D" )
   END_RUNG wire#w1
   RUNG wire#powerrail
      Contact( "FALLAS HMI"."FALLA BREAKER Q5 - VFD 5 096P001E" )
   END_RUNG wire#w1
   RUNG wire#powerrail
      Contact( "FALLAS HMI"."FALLA VARIADOR VELOCIDAD 096P001E" )
   END_RUNG wire#w1
   RUNG wire#powerrail
      Contact( "FALLAS HMI"."PARO DE EMERGENCIA ACTIVO 096P001E" )
   END_RUNG wire#w1
   RUNG wire#powerrail
      Contact( "FALLAS HMI"."NO CONFIRMA ARRANQUE BOMBA 096P001E" )
   END_RUNG wire#w1
   RUNG wire#powerrail
      Contact( "FALLAS HMI"."FALLA BREAKER Q6 - VFD 6 096P001F" )
   END_RUNG wire#w1
   RUNG wire#powerrail
      Contact( "FALLAS HMI"."FALLA VARIADOR VELOCIDAD 096P001F" )
   END_RUNG wire#w1
   RUNG wire#powerrail
      Contact( "FALLAS HMI"."PARO DE EMERGENCIA ACTIVO 096P001F" )
   END_RUNG wire#w1
   RUNG wire#powerrail
      Contact( "FALLAS HMI"."NO CONFIRMA ARRANQUE BOMBA 096P001F" )
   END_RUNG wire#w1
   RUNG wire#powerrail
      Contact( "FALLAS HMI"."SWITCH DE PRESION EN SUCCION INACTIVO PSL001" )
   END_RUNG wire#w1
   RUNG wire#powerrail
      Contact( "FALLAS HMI"."SWITCH DE FLUJO EN SUCCION INACTIVO FSL001" )
   END_RUNG wire#w1
   RUNG wire#powerrail
      Contact( "FALLAS HMI"."NO CONFIRMA SWITCH DE FLUJO CON BOMBA 096P001A" )
   END_RUNG wire#w1
   RUNG wire#powerrail
      Contact( "FALLAS HMI"."NO CONFIRMA SWITCH DE FLUJO CON BOMBA 096P001B" )
   END_RUNG wire#w1
   RUNG wire#powerrail
      Contact( "FALLAS HMI"."NO CONFIRMA SWITCH DE FLUJO CON BOMBA 096P001C" )
   END_RUNG wire#w1
   RUNG wire#powerrail
      Contact( "FALLAS HMI"."NO CONFIRMA SWITCH DE FLUJO CON BOMBA 096P001D" )
   END_RUNG wire#w1
   RUNG wire#powerrail
      Contact( "FALLAS HMI"."NO CONFIRMA SWITCH DE FLUJO CON BOMBA 096P001E" )
   END_RUNG wire#w1
   RUNG wire#powerrail
      Contact( "FALLAS HMI"."NO CONFIRMA SWITCH DE FLUJO CON BOMBA 096P001F" )
   END_RUNG wire#w1
   RUNG wire#powerrail
      Contact( "FALLAS HMI"."FALLA POR ALTA PRESION DE DESCARGA 096PIT002" )
   END_RUNG wire#w1
   RUNG wire#powerrail
      Contact( "FALLAS HMI"."ALARMA POR ALTA PRESION DE DESCARGA 096PIT002" )
   END_RUNG wire#w1
   RUNG wire#powerrail
      Contact( "FALLAS HMI"."ALARMA POR BAJA PRESION DE DESCARGA 096PIT002" )
   END_RUNG wire#w1
   RUNG wire#powerrail
      Contact( "FALLAS HMI"."FALLA POR BAJA PRESION DE DESCARGA 096PIT002" )
   END_RUNG wire#w1
   RUNG wire#powerrail
      Contact( "FALLAS HMI"."FALLA POR ALTA PRESION DE SUCCION 096PIT001" )
   END_RUNG wire#w1
   RUNG wire#powerrail
      Contact( "FALLAS HMI"."ALARMA POR ALTA PRESION DE SUCCION 096PIT001" )
   END_RUNG wire#w1
   RUNG wire#powerrail
      Contact( "FALLAS HMI"."ALARMA POR BAJA PRESION DE SUCCION 096PIT001" )
   END_RUNG wire#w1
   RUNG wire#powerrail
      Contact( "FALLAS HMI"."FALLA POR BAJA PRESION DE SUCCION 096PIT001" )
   END_RUNG wire#w1
   // the same network as SCL:
   "Alarmas Sis servicio"."Alarma general" := "FALLAS HMI"."PARO EMERGENCIA ACTIVO SISTEMA GRAL AGUA SERVICIO" OR "FALLAS HMI"."FALLA BREAKER PRINCIPAL" OR "FALLAS HMI"."FALLA BREAKER Q1 - VFD 1 096P001A" OR "FALLAS HMI"."FALLA VARIADOR VELOCIDAD 096P001A" OR "FALLAS HMI"."PARO DE EMERGENCIA ACTIVO 096P001A" OR "FALLAS HMI"."NO CONFIRMA ARRANQUE BOMBA 096P001A" OR "FALLAS HMI"."FALLA BREAKER Q2 - VFD 2 096P001B" OR "FALLAS HMI"."FALLA VARIADOR VELOCIDAD 096P001B" OR "FALLAS HMI"."PARO DE EMERGENCIA ACTIVO 096P001B" OR "FALLAS HMI"."NO CONFIRMA ARRANQUE BOMBA 096P001B" OR "FALLAS HMI"."FALLA BREAKER Q3 - VFD 3 096P001C" OR "FALLAS HMI"."FALLA VARIADOR VELOCIDAD 096P001C" OR "FALLAS HMI"."PARO DE EMERGENCIA ACTIVO 096P001C" OR "FALLAS HMI"."NO CONFIRMA ARRANQUE BOMBA 096P001C" OR "FALLAS HMI"."FALLA BREAKER Q4 - VFD 4 096P001D" OR "FALLAS HMI"."FALLA VARIADOR VELOCIDAD 096P001D" OR "FALLAS HMI"."PARO DE EMERGENCIA ACTIVO 096P001D" OR "FALLAS HMI"."NO CONFIRMA ARRANQUE BOMBA 096P001D" OR "FALLAS HMI"."FALLA BREAKER Q5 - VFD 5 096P001E" OR "FALLAS HMI"."FALLA VARIADOR VELOCIDAD 096P001E" OR "FALLAS HMI"."PARO DE EMERGENCIA ACTIVO 096P001E" OR "FALLAS HMI"."NO CONFIRMA ARRANQUE BOMBA 096P001E" OR "FALLAS HMI"."FALLA BREAKER Q6 - VFD 6 096P001F" OR "FALLAS HMI"."FALLA VARIADOR VELOCIDAD 096P001F" OR "FALLAS HMI"."PARO DE EMERGENCIA ACTIVO 096P001F" OR "FALLAS HMI"."NO CONFIRMA ARRANQUE BOMBA 096P001F" OR "FALLAS HMI"."SWITCH DE PRESION EN SUCCION INACTIVO PSL001" OR "FALLAS HMI"."SWITCH DE FLUJO EN SUCCION INACTIVO FSL001" OR "FALLAS HMI"."NO CONFIRMA SWITCH DE FLUJO CON BOMBA 096P001A" OR "FALLAS HMI"."NO CONFIRMA SWITCH DE FLUJO CON BOMBA 096P001B" OR "FALLAS HMI"."NO CONFIRMA SWITCH DE FLUJO CON BOMBA 096P001C" OR "FALLAS HMI"."NO CONFIRMA SWITCH DE FLUJO CON BOMBA 096P001D" OR "FALLAS HMI"."NO CONFIRMA SWITCH DE FLUJO CON BOMBA 096P001E" OR "FALLAS HMI"."NO CONFIRMA SWITCH DE FLUJO CON BOMBA 096P001F" OR "FALLAS HMI"."FALLA POR ALTA PRESION DE DESCARGA 096PIT002" OR "FALLAS HMI"."ALARMA POR ALTA PRESION DE DESCARGA 096PIT002" OR "FALLAS HMI"."ALARMA POR BAJA PRESION DE DESCARGA 096PIT002" OR "FALLAS HMI"."FALLA POR BAJA PRESION DE DESCARGA 096PIT002" OR "FALLAS HMI"."FALLA POR ALTA PRESION DE SUCCION 096PIT001" OR "FALLAS HMI"."ALARMA POR ALTA PRESION DE SUCCION 096PIT001" OR "FALLAS HMI"."ALARMA POR BAJA PRESION DE SUCCION 096PIT001" OR "FALLAS HMI"."FALLA POR BAJA PRESION DE SUCCION 096PIT001";
END_REGION
END_FUNCTION

FUNCTION "Esc Salidas Analogas" : Void   // FC12, LAD
{ S7_Optimized_Access := 'TRUE' }
VERSION : 0.1
   VAR_TEMP
      SA1 : Real;
      SA2 : Real;
      SA3 : Real;
      SA4 : Real;
      SA5 : Real;
      SA6 : Real;
      "CONSIGNA 1" : Real;
      "CONSIGNA 2" : Real;
      "CONSIGNA 3" : Real;
      "CONSIGNA 4" : Real;
      "CONSIGNA 5" : Real;
      "CONSIGNA 6" : Real;
   END_VAR
BEGIN

REGION Network 1: SALIDA ANALOGA 096P001A
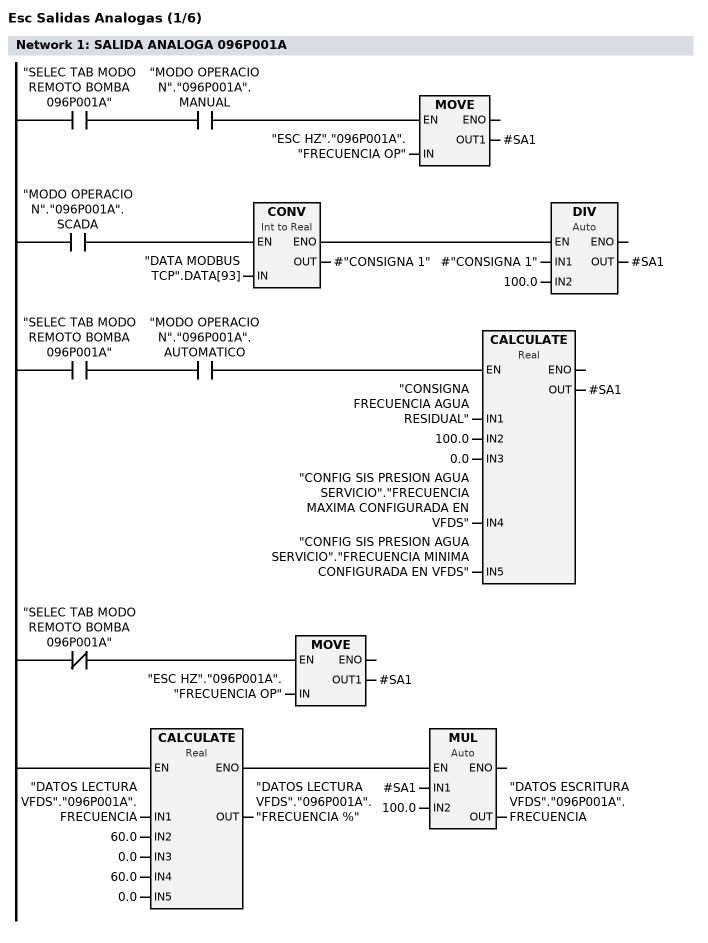
   RUNG wire#powerrail
      Contact( "SELEC TAB MODO REMOTO BOMBA 096P001A" )
      Contact( "MODO OPERACION"."096P001A".MANUAL )
      Move(in := "ESC HZ"."096P001A"."FRECUENCIA OP", out1 => #SA1)
   END_RUNG
   RUNG wire#powerrail
      Contact( "MODO OPERACION"."096P001A".SCADA )
      { S7_Templates := "[SrcType := Int, DestType := Real]" } Convert(in := "DATA MODBUS TCP".DATA[93], out => #"CONSIGNA 1")
      Div(in1 := #"CONSIGNA 1", in2 := 100.0, out => #SA1)
   END_RUNG
   RUNG wire#powerrail
      Contact( "SELEC TAB MODO REMOTO BOMBA 096P001A" )
      Contact( "MODO OPERACION"."096P001A".AUTOMATICO )
      { S7_Templates := "SrcType := Real"; S7_Expression := "(((IN4-IN5)/(IN2-IN3))*IN1)+(IN5-(((IN4-IN5)/(IN2-IN3))*IN3))" } Calculate(in1 := "CONSIGNA FRECUENCIA AGUA RESIDUAL", in2 := 100.0, in3 := 0.0, in4 := "CONFIG SIS PRESION AGUA SERVICIO"."FRECUENCIA MAXIMA CONFIGURADA EN VFDS", in5 := "CONFIG SIS PRESION AGUA SERVICIO"."FRECUENCIA MINIMA CONFIGURADA EN VFDS", out => #SA1)
   END_RUNG
   RUNG wire#powerrail
      I_Contact( "SELEC TAB MODO REMOTO BOMBA 096P001A" )
      Move(in := "ESC HZ"."096P001A"."FRECUENCIA OP", out1 => #SA1)
   END_RUNG
   RUNG wire#powerrail
      { S7_Templates := "SrcType := Real"; S7_Expression := "(((IN4-IN5)/(IN2-IN3))*IN1)+(IN5-(((IN4-IN5)/(IN2-IN3))*IN3))" } Calculate(in1 := "DATOS LECTURA VFDS"."096P001A".FRECUENCIA, in2 := 60.0, in3 := 0.0, in4 := 60.0, in5 := 0.0, out => "DATOS LECTURA VFDS"."096P001A"."FRECUENCIA %")
      Mul(in1 := #SA1, in2 := 100.0, out => "DATOS ESCRITURA VFDS"."096P001A".FRECUENCIA)
   END_RUNG
   // the same network as SCL:
   IF "SELEC TAB MODO REMOTO BOMBA 096P001A" AND "MODO OPERACION"."096P001A".MANUAL THEN
       #SA1 := "ESC HZ"."096P001A"."FRECUENCIA OP";
   END_IF;
   IF "MODO OPERACION"."096P001A".SCADA THEN
       #"CONSIGNA 1" := INT_TO_REAL("DATA MODBUS TCP".DATA[93]);
       #SA1 := #"CONSIGNA 1" / 100.0;
   END_IF;
   IF "SELEC TAB MODO REMOTO BOMBA 096P001A" AND "MODO OPERACION"."096P001A".AUTOMATICO THEN
       #SA1 := ((("CONFIG SIS PRESION AGUA SERVICIO"."FRECUENCIA MAXIMA CONFIGURADA EN VFDS"-"CONFIG SIS PRESION AGUA SERVICIO"."FRECUENCIA MINIMA CONFIGURADA EN VFDS")/(100.0-0.0))*"CONSIGNA FRECUENCIA AGUA RESIDUAL")+("CONFIG SIS PRESION AGUA SERVICIO"."FRECUENCIA MINIMA CONFIGURADA EN VFDS"-((("CONFIG SIS PRESION AGUA SERVICIO"."FRECUENCIA MAXIMA CONFIGURADA EN VFDS"-"CONFIG SIS PRESION AGUA SERVICIO"."FRECUENCIA MINIMA CONFIGURADA EN VFDS")/(100.0-0.0))*0.0));
   END_IF;
   IF NOT "SELEC TAB MODO REMOTO BOMBA 096P001A" THEN #SA1 := "ESC HZ"."096P001A"."FRECUENCIA OP"; END_IF;
   "DATOS LECTURA VFDS"."096P001A"."FRECUENCIA %" := (((60.0-0.0)/(60.0-0.0))*"DATOS LECTURA VFDS"."096P001A".FRECUENCIA)+(0.0-(((60.0-0.0)/(60.0-0.0))*0.0));
   "DATOS ESCRITURA VFDS"."096P001A".FRECUENCIA := #SA1 * 100.0;
END_REGION

REGION Network 2: SALIDA ANALOGA 096P001B
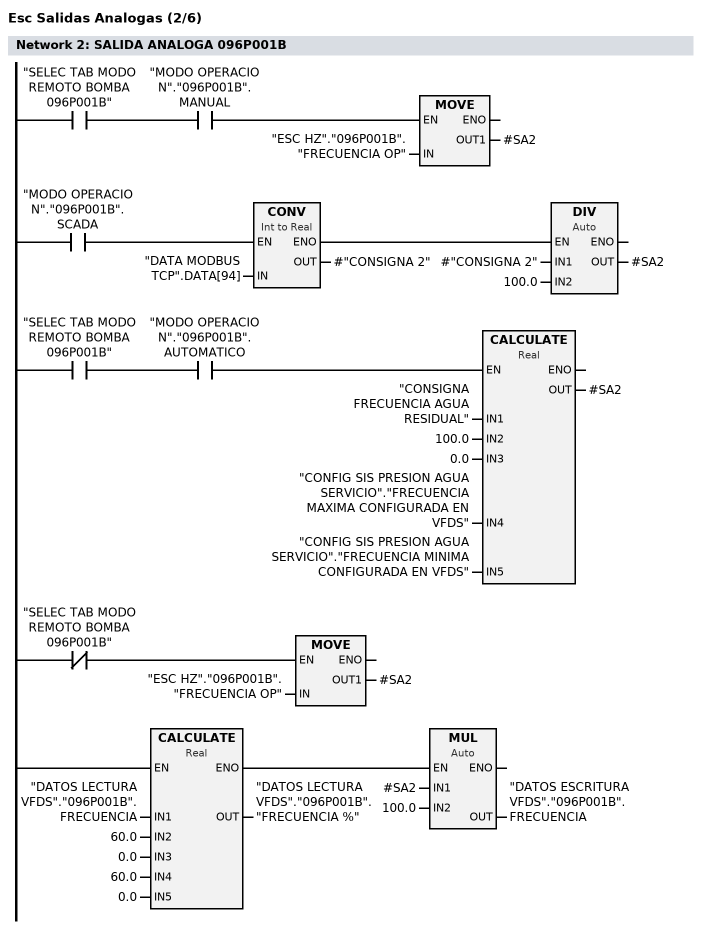
   RUNG wire#powerrail
      Contact( "SELEC TAB MODO REMOTO BOMBA 096P001B" )
      Contact( "MODO OPERACION"."096P001B".MANUAL )
      Move(in := "ESC HZ"."096P001B"."FRECUENCIA OP", out1 => #SA2)
   END_RUNG
   RUNG wire#powerrail
      Contact( "MODO OPERACION"."096P001B".SCADA )
      { S7_Templates := "[SrcType := Int, DestType := Real]" } Convert(in := "DATA MODBUS TCP".DATA[94], out => #"CONSIGNA 2")
      Div(in1 := #"CONSIGNA 2", in2 := 100.0, out => #SA2)
   END_RUNG
   RUNG wire#powerrail
      Contact( "SELEC TAB MODO REMOTO BOMBA 096P001B" )
      Contact( "MODO OPERACION"."096P001B".AUTOMATICO )
      { S7_Templates := "SrcType := Real"; S7_Expression := "(((IN4-IN5)/(IN2-IN3))*IN1)+(IN5-(((IN4-IN5)/(IN2-IN3))*IN3))" } Calculate(in1 := "CONSIGNA FRECUENCIA AGUA RESIDUAL", in2 := 100.0, in3 := 0.0, in4 := "CONFIG SIS PRESION AGUA SERVICIO"."FRECUENCIA MAXIMA CONFIGURADA EN VFDS", in5 := "CONFIG SIS PRESION AGUA SERVICIO"."FRECUENCIA MINIMA CONFIGURADA EN VFDS", out => #SA2)
   END_RUNG
   RUNG wire#powerrail
      I_Contact( "SELEC TAB MODO REMOTO BOMBA 096P001B" )
      Move(in := "ESC HZ"."096P001B"."FRECUENCIA OP", out1 => #SA2)
   END_RUNG
   RUNG wire#powerrail
      { S7_Templates := "SrcType := Real"; S7_Expression := "(((IN4-IN5)/(IN2-IN3))*IN1)+(IN5-(((IN4-IN5)/(IN2-IN3))*IN3))" } Calculate(in1 := "DATOS LECTURA VFDS"."096P001B".FRECUENCIA, in2 := 60.0, in3 := 0.0, in4 := 60.0, in5 := 0.0, out => "DATOS LECTURA VFDS"."096P001B"."FRECUENCIA %")
      Mul(in1 := #SA2, in2 := 100.0, out => "DATOS ESCRITURA VFDS"."096P001B".FRECUENCIA)
   END_RUNG
   // the same network as SCL:
   IF "SELEC TAB MODO REMOTO BOMBA 096P001B" AND "MODO OPERACION"."096P001B".MANUAL THEN
       #SA2 := "ESC HZ"."096P001B"."FRECUENCIA OP";
   END_IF;
   IF "MODO OPERACION"."096P001B".SCADA THEN
       #"CONSIGNA 2" := INT_TO_REAL("DATA MODBUS TCP".DATA[94]);
       #SA2 := #"CONSIGNA 2" / 100.0;
   END_IF;
   IF "SELEC TAB MODO REMOTO BOMBA 096P001B" AND "MODO OPERACION"."096P001B".AUTOMATICO THEN
       #SA2 := ((("CONFIG SIS PRESION AGUA SERVICIO"."FRECUENCIA MAXIMA CONFIGURADA EN VFDS"-"CONFIG SIS PRESION AGUA SERVICIO"."FRECUENCIA MINIMA CONFIGURADA EN VFDS")/(100.0-0.0))*"CONSIGNA FRECUENCIA AGUA RESIDUAL")+("CONFIG SIS PRESION AGUA SERVICIO"."FRECUENCIA MINIMA CONFIGURADA EN VFDS"-((("CONFIG SIS PRESION AGUA SERVICIO"."FRECUENCIA MAXIMA CONFIGURADA EN VFDS"-"CONFIG SIS PRESION AGUA SERVICIO"."FRECUENCIA MINIMA CONFIGURADA EN VFDS")/(100.0-0.0))*0.0));
   END_IF;
   IF NOT "SELEC TAB MODO REMOTO BOMBA 096P001B" THEN #SA2 := "ESC HZ"."096P001B"."FRECUENCIA OP"; END_IF;
   "DATOS LECTURA VFDS"."096P001B"."FRECUENCIA %" := (((60.0-0.0)/(60.0-0.0))*"DATOS LECTURA VFDS"."096P001B".FRECUENCIA)+(0.0-(((60.0-0.0)/(60.0-0.0))*0.0));
   "DATOS ESCRITURA VFDS"."096P001B".FRECUENCIA := #SA2 * 100.0;
END_REGION

REGION Network 3: SALIDA ANALOGA 096P001C
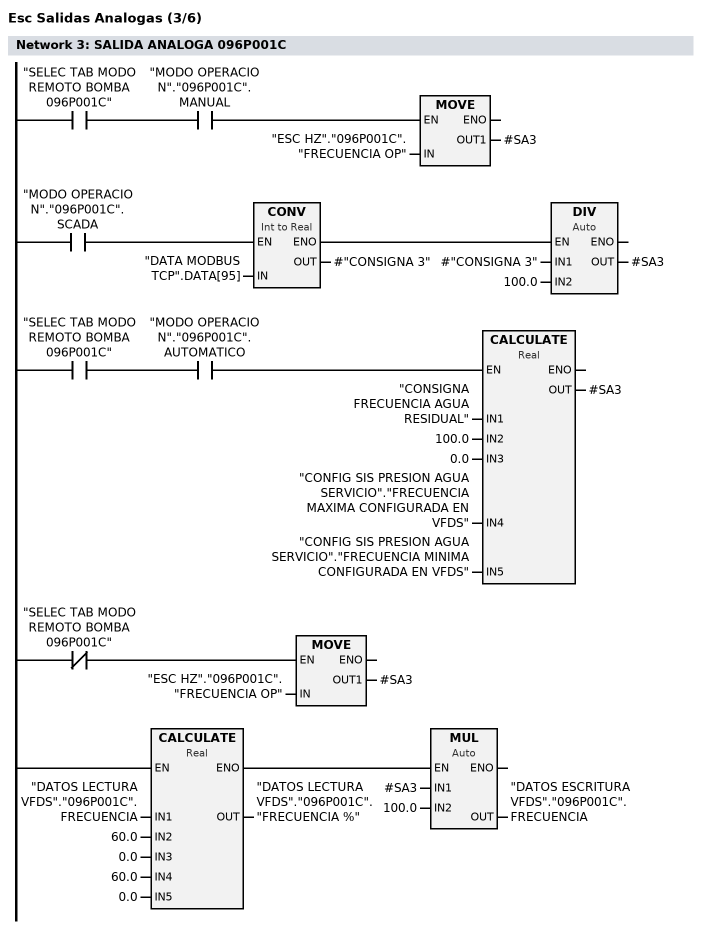
   RUNG wire#powerrail
      Contact( "SELEC TAB MODO REMOTO BOMBA 096P001C" )
      Contact( "MODO OPERACION"."096P001C".MANUAL )
      Move(in := "ESC HZ"."096P001C"."FRECUENCIA OP", out1 => #SA3)
   END_RUNG
   RUNG wire#powerrail
      Contact( "MODO OPERACION"."096P001C".SCADA )
      { S7_Templates := "[SrcType := Int, DestType := Real]" } Convert(in := "DATA MODBUS TCP".DATA[95], out => #"CONSIGNA 3")
      Div(in1 := #"CONSIGNA 3", in2 := 100.0, out => #SA3)
   END_RUNG
   RUNG wire#powerrail
      Contact( "SELEC TAB MODO REMOTO BOMBA 096P001C" )
      Contact( "MODO OPERACION"."096P001C".AUTOMATICO )
      { S7_Templates := "SrcType := Real"; S7_Expression := "(((IN4-IN5)/(IN2-IN3))*IN1)+(IN5-(((IN4-IN5)/(IN2-IN3))*IN3))" } Calculate(in1 := "CONSIGNA FRECUENCIA AGUA RESIDUAL", in2 := 100.0, in3 := 0.0, in4 := "CONFIG SIS PRESION AGUA SERVICIO"."FRECUENCIA MAXIMA CONFIGURADA EN VFDS", in5 := "CONFIG SIS PRESION AGUA SERVICIO"."FRECUENCIA MINIMA CONFIGURADA EN VFDS", out => #SA3)
   END_RUNG
   RUNG wire#powerrail
      I_Contact( "SELEC TAB MODO REMOTO BOMBA 096P001C" )
      Move(in := "ESC HZ"."096P001C"."FRECUENCIA OP", out1 => #SA3)
   END_RUNG
   RUNG wire#powerrail
      { S7_Templates := "SrcType := Real"; S7_Expression := "(((IN4-IN5)/(IN2-IN3))*IN1)+(IN5-(((IN4-IN5)/(IN2-IN3))*IN3))" } Calculate(in1 := "DATOS LECTURA VFDS"."096P001C".FRECUENCIA, in2 := 60.0, in3 := 0.0, in4 := 60.0, in5 := 0.0, out => "DATOS LECTURA VFDS"."096P001C"."FRECUENCIA %")
      Mul(in1 := #SA3, in2 := 100.0, out => "DATOS ESCRITURA VFDS"."096P001C".FRECUENCIA)
   END_RUNG
   // the same network as SCL:
   IF "SELEC TAB MODO REMOTO BOMBA 096P001C" AND "MODO OPERACION"."096P001C".MANUAL THEN
       #SA3 := "ESC HZ"."096P001C"."FRECUENCIA OP";
   END_IF;
   IF "MODO OPERACION"."096P001C".SCADA THEN
       #"CONSIGNA 3" := INT_TO_REAL("DATA MODBUS TCP".DATA[95]);
       #SA3 := #"CONSIGNA 3" / 100.0;
   END_IF;
   IF "SELEC TAB MODO REMOTO BOMBA 096P001C" AND "MODO OPERACION"."096P001C".AUTOMATICO THEN
       #SA3 := ((("CONFIG SIS PRESION AGUA SERVICIO"."FRECUENCIA MAXIMA CONFIGURADA EN VFDS"-"CONFIG SIS PRESION AGUA SERVICIO"."FRECUENCIA MINIMA CONFIGURADA EN VFDS")/(100.0-0.0))*"CONSIGNA FRECUENCIA AGUA RESIDUAL")+("CONFIG SIS PRESION AGUA SERVICIO"."FRECUENCIA MINIMA CONFIGURADA EN VFDS"-((("CONFIG SIS PRESION AGUA SERVICIO"."FRECUENCIA MAXIMA CONFIGURADA EN VFDS"-"CONFIG SIS PRESION AGUA SERVICIO"."FRECUENCIA MINIMA CONFIGURADA EN VFDS")/(100.0-0.0))*0.0));
   END_IF;
   IF NOT "SELEC TAB MODO REMOTO BOMBA 096P001C" THEN #SA3 := "ESC HZ"."096P001C"."FRECUENCIA OP"; END_IF;
   "DATOS LECTURA VFDS"."096P001C"."FRECUENCIA %" := (((60.0-0.0)/(60.0-0.0))*"DATOS LECTURA VFDS"."096P001C".FRECUENCIA)+(0.0-(((60.0-0.0)/(60.0-0.0))*0.0));
   "DATOS ESCRITURA VFDS"."096P001C".FRECUENCIA := #SA3 * 100.0;
END_REGION

REGION Network 4: SALIDA ANALOGA 096P001D
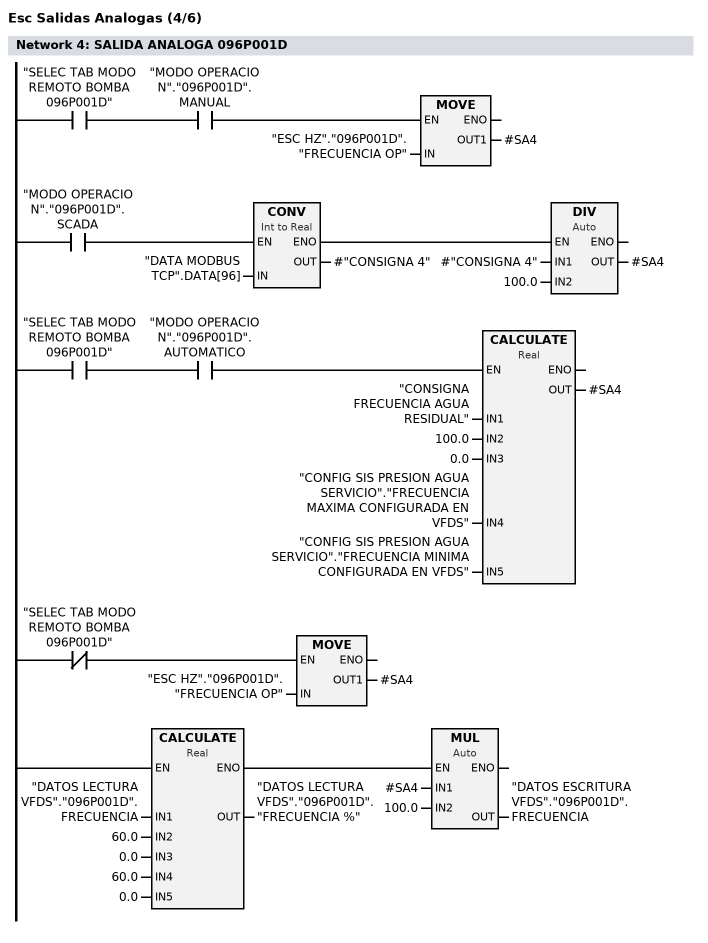
   RUNG wire#powerrail
      Contact( "SELEC TAB MODO REMOTO BOMBA 096P001D" )
      Contact( "MODO OPERACION"."096P001D".MANUAL )
      Move(in := "ESC HZ"."096P001D"."FRECUENCIA OP", out1 => #SA4)
   END_RUNG
   RUNG wire#powerrail
      Contact( "MODO OPERACION"."096P001D".SCADA )
      { S7_Templates := "[SrcType := Int, DestType := Real]" } Convert(in := "DATA MODBUS TCP".DATA[96], out => #"CONSIGNA 4")
      Div(in1 := #"CONSIGNA 4", in2 := 100.0, out => #SA4)
   END_RUNG
   RUNG wire#powerrail
      Contact( "SELEC TAB MODO REMOTO BOMBA 096P001D" )
      Contact( "MODO OPERACION"."096P001D".AUTOMATICO )
      { S7_Templates := "SrcType := Real"; S7_Expression := "(((IN4-IN5)/(IN2-IN3))*IN1)+(IN5-(((IN4-IN5)/(IN2-IN3))*IN3))" } Calculate(in1 := "CONSIGNA FRECUENCIA AGUA RESIDUAL", in2 := 100.0, in3 := 0.0, in4 := "CONFIG SIS PRESION AGUA SERVICIO"."FRECUENCIA MAXIMA CONFIGURADA EN VFDS", in5 := "CONFIG SIS PRESION AGUA SERVICIO"."FRECUENCIA MINIMA CONFIGURADA EN VFDS", out => #SA4)
   END_RUNG
   RUNG wire#powerrail
      I_Contact( "SELEC TAB MODO REMOTO BOMBA 096P001D" )
      Move(in := "ESC HZ"."096P001D"."FRECUENCIA OP", out1 => #SA4)
   END_RUNG
   RUNG wire#powerrail
      { S7_Templates := "SrcType := Real"; S7_Expression := "(((IN4-IN5)/(IN2-IN3))*IN1)+(IN5-(((IN4-IN5)/(IN2-IN3))*IN3))" } Calculate(in1 := "DATOS LECTURA VFDS"."096P001D".FRECUENCIA, in2 := 60.0, in3 := 0.0, in4 := 60.0, in5 := 0.0, out => "DATOS LECTURA VFDS"."096P001D"."FRECUENCIA %")
      Mul(in1 := #SA4, in2 := 100.0, out => "DATOS ESCRITURA VFDS"."096P001D".FRECUENCIA)
   END_RUNG
   // the same network as SCL:
   IF "SELEC TAB MODO REMOTO BOMBA 096P001D" AND "MODO OPERACION"."096P001D".MANUAL THEN
       #SA4 := "ESC HZ"."096P001D"."FRECUENCIA OP";
   END_IF;
   IF "MODO OPERACION"."096P001D".SCADA THEN
       #"CONSIGNA 4" := INT_TO_REAL("DATA MODBUS TCP".DATA[96]);
       #SA4 := #"CONSIGNA 4" / 100.0;
   END_IF;
   IF "SELEC TAB MODO REMOTO BOMBA 096P001D" AND "MODO OPERACION"."096P001D".AUTOMATICO THEN
       #SA4 := ((("CONFIG SIS PRESION AGUA SERVICIO"."FRECUENCIA MAXIMA CONFIGURADA EN VFDS"-"CONFIG SIS PRESION AGUA SERVICIO"."FRECUENCIA MINIMA CONFIGURADA EN VFDS")/(100.0-0.0))*"CONSIGNA FRECUENCIA AGUA RESIDUAL")+("CONFIG SIS PRESION AGUA SERVICIO"."FRECUENCIA MINIMA CONFIGURADA EN VFDS"-((("CONFIG SIS PRESION AGUA SERVICIO"."FRECUENCIA MAXIMA CONFIGURADA EN VFDS"-"CONFIG SIS PRESION AGUA SERVICIO"."FRECUENCIA MINIMA CONFIGURADA EN VFDS")/(100.0-0.0))*0.0));
   END_IF;
   IF NOT "SELEC TAB MODO REMOTO BOMBA 096P001D" THEN #SA4 := "ESC HZ"."096P001D"."FRECUENCIA OP"; END_IF;
   "DATOS LECTURA VFDS"."096P001D"."FRECUENCIA %" := (((60.0-0.0)/(60.0-0.0))*"DATOS LECTURA VFDS"."096P001D".FRECUENCIA)+(0.0-(((60.0-0.0)/(60.0-0.0))*0.0));
   "DATOS ESCRITURA VFDS"."096P001D".FRECUENCIA := #SA4 * 100.0;
END_REGION

REGION Network 5: SALIDA ANALOGA 096P001E
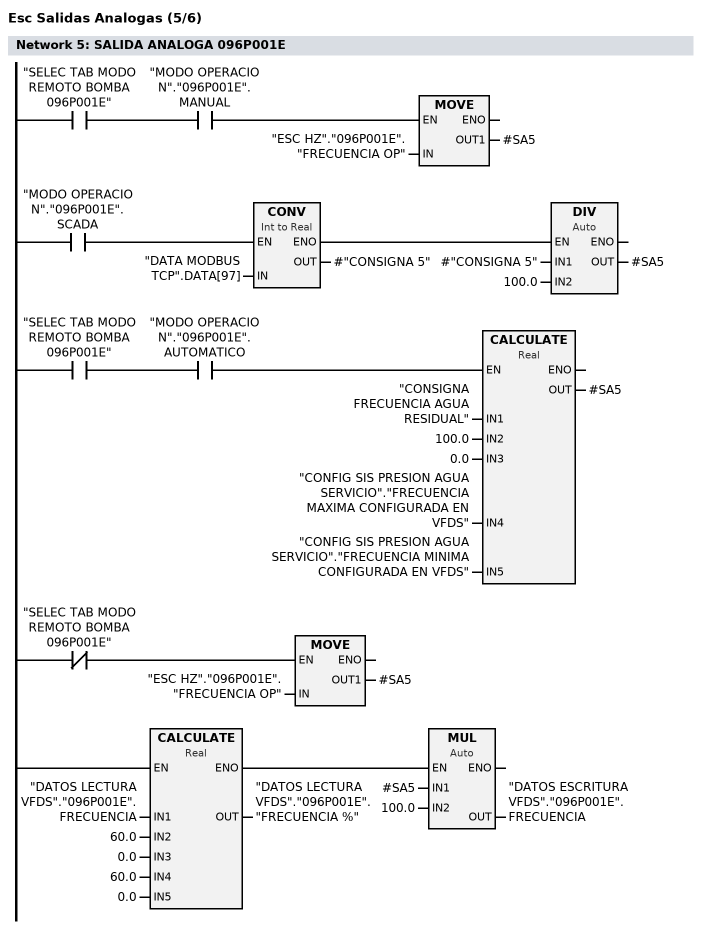
   RUNG wire#powerrail
      Contact( "SELEC TAB MODO REMOTO BOMBA 096P001E" )
      Contact( "MODO OPERACION"."096P001E".MANUAL )
      Move(in := "ESC HZ"."096P001E"."FRECUENCIA OP", out1 => #SA5)
   END_RUNG
   RUNG wire#powerrail
      Contact( "MODO OPERACION"."096P001E".SCADA )
      { S7_Templates := "[SrcType := Int, DestType := Real]" } Convert(in := "DATA MODBUS TCP".DATA[97], out => #"CONSIGNA 5")
      Div(in1 := #"CONSIGNA 5", in2 := 100.0, out => #SA5)
   END_RUNG
   RUNG wire#powerrail
      Contact( "SELEC TAB MODO REMOTO BOMBA 096P001E" )
      Contact( "MODO OPERACION"."096P001E".AUTOMATICO )
      { S7_Templates := "SrcType := Real"; S7_Expression := "(((IN4-IN5)/(IN2-IN3))*IN1)+(IN5-(((IN4-IN5)/(IN2-IN3))*IN3))" } Calculate(in1 := "CONSIGNA FRECUENCIA AGUA RESIDUAL", in2 := 100.0, in3 := 0.0, in4 := "CONFIG SIS PRESION AGUA SERVICIO"."FRECUENCIA MAXIMA CONFIGURADA EN VFDS", in5 := "CONFIG SIS PRESION AGUA SERVICIO"."FRECUENCIA MINIMA CONFIGURADA EN VFDS", out => #SA5)
   END_RUNG
   RUNG wire#powerrail
      I_Contact( "SELEC TAB MODO REMOTO BOMBA 096P001E" )
      Move(in := "ESC HZ"."096P001E"."FRECUENCIA OP", out1 => #SA5)
   END_RUNG
   RUNG wire#powerrail
      { S7_Templates := "SrcType := Real"; S7_Expression := "(((IN4-IN5)/(IN2-IN3))*IN1)+(IN5-(((IN4-IN5)/(IN2-IN3))*IN3))" } Calculate(in1 := "DATOS LECTURA VFDS"."096P001E".FRECUENCIA, in2 := 60.0, in3 := 0.0, in4 := 60.0, in5 := 0.0, out => "DATOS LECTURA VFDS"."096P001E"."FRECUENCIA %")
      Mul(in1 := #SA5, in2 := 100.0, out => "DATOS ESCRITURA VFDS"."096P001E".FRECUENCIA)
   END_RUNG
   // the same network as SCL:
   IF "SELEC TAB MODO REMOTO BOMBA 096P001E" AND "MODO OPERACION"."096P001E".MANUAL THEN
       #SA5 := "ESC HZ"."096P001E"."FRECUENCIA OP";
   END_IF;
   IF "MODO OPERACION"."096P001E".SCADA THEN
       #"CONSIGNA 5" := INT_TO_REAL("DATA MODBUS TCP".DATA[97]);
       #SA5 := #"CONSIGNA 5" / 100.0;
   END_IF;
   IF "SELEC TAB MODO REMOTO BOMBA 096P001E" AND "MODO OPERACION"."096P001E".AUTOMATICO THEN
       #SA5 := ((("CONFIG SIS PRESION AGUA SERVICIO"."FRECUENCIA MAXIMA CONFIGURADA EN VFDS"-"CONFIG SIS PRESION AGUA SERVICIO"."FRECUENCIA MINIMA CONFIGURADA EN VFDS")/(100.0-0.0))*"CONSIGNA FRECUENCIA AGUA RESIDUAL")+("CONFIG SIS PRESION AGUA SERVICIO"."FRECUENCIA MINIMA CONFIGURADA EN VFDS"-((("CONFIG SIS PRESION AGUA SERVICIO"."FRECUENCIA MAXIMA CONFIGURADA EN VFDS"-"CONFIG SIS PRESION AGUA SERVICIO"."FRECUENCIA MINIMA CONFIGURADA EN VFDS")/(100.0-0.0))*0.0));
   END_IF;
   IF NOT "SELEC TAB MODO REMOTO BOMBA 096P001E" THEN #SA5 := "ESC HZ"."096P001E"."FRECUENCIA OP"; END_IF;
   "DATOS LECTURA VFDS"."096P001E"."FRECUENCIA %" := (((60.0-0.0)/(60.0-0.0))*"DATOS LECTURA VFDS"."096P001E".FRECUENCIA)+(0.0-(((60.0-0.0)/(60.0-0.0))*0.0));
   "DATOS ESCRITURA VFDS"."096P001E".FRECUENCIA := #SA5 * 100.0;
END_REGION

REGION Network 6: SALIDA ANALOGA 096P001F
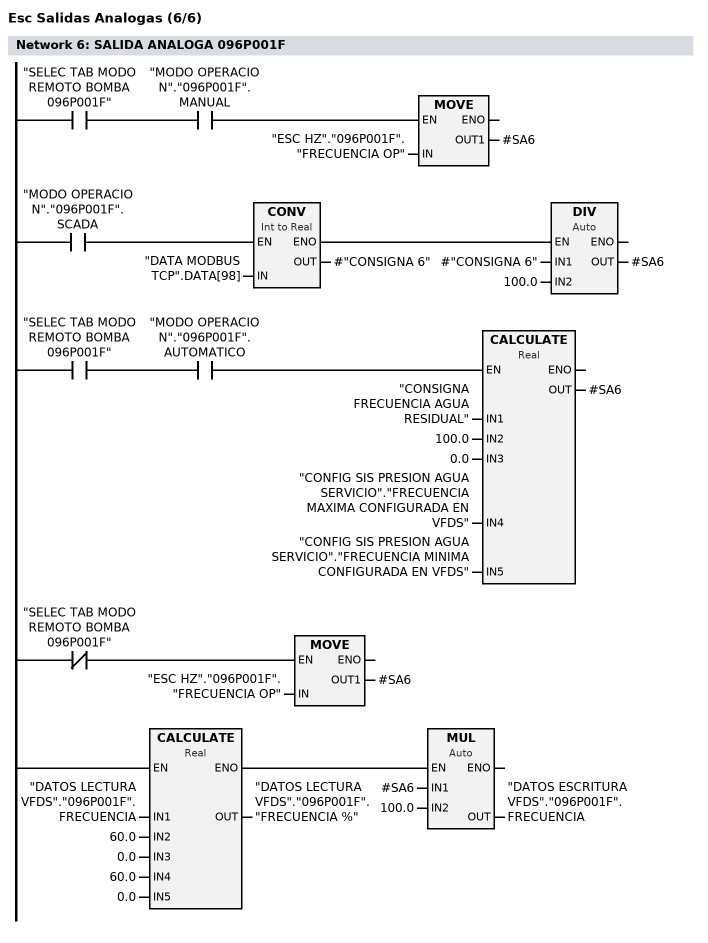
   RUNG wire#powerrail
      Contact( "SELEC TAB MODO REMOTO BOMBA 096P001F" )
      Contact( "MODO OPERACION"."096P001F".MANUAL )
      Move(in := "ESC HZ"."096P001F"."FRECUENCIA OP", out1 => #SA6)
   END_RUNG
   RUNG wire#powerrail
      Contact( "MODO OPERACION"."096P001F".SCADA )
      { S7_Templates := "[SrcType := Int, DestType := Real]" } Convert(in := "DATA MODBUS TCP".DATA[98], out => #"CONSIGNA 6")
      Div(in1 := #"CONSIGNA 6", in2 := 100.0, out => #SA6)
   END_RUNG
   RUNG wire#powerrail
      Contact( "SELEC TAB MODO REMOTO BOMBA 096P001F" )
      Contact( "MODO OPERACION"."096P001F".AUTOMATICO )
      { S7_Templates := "SrcType := Real"; S7_Expression := "(((IN4-IN5)/(IN2-IN3))*IN1)+(IN5-(((IN4-IN5)/(IN2-IN3))*IN3))" } Calculate(in1 := "CONSIGNA FRECUENCIA AGUA RESIDUAL", in2 := 100.0, in3 := 0.0, in4 := "CONFIG SIS PRESION AGUA SERVICIO"."FRECUENCIA MAXIMA CONFIGURADA EN VFDS", in5 := "CONFIG SIS PRESION AGUA SERVICIO"."FRECUENCIA MINIMA CONFIGURADA EN VFDS", out => #SA6)
   END_RUNG
   RUNG wire#powerrail
      I_Contact( "SELEC TAB MODO REMOTO BOMBA 096P001F" )
      Move(in := "ESC HZ"."096P001F"."FRECUENCIA OP", out1 => #SA6)
   END_RUNG
   RUNG wire#powerrail
      { S7_Templates := "SrcType := Real"; S7_Expression := "(((IN4-IN5)/(IN2-IN3))*IN1)+(IN5-(((IN4-IN5)/(IN2-IN3))*IN3))" } Calculate(in1 := "DATOS LECTURA VFDS"."096P001F".FRECUENCIA, in2 := 60.0, in3 := 0.0, in4 := 60.0, in5 := 0.0, out => "DATOS LECTURA VFDS"."096P001F"."FRECUENCIA %")
      Mul(in1 := #SA6, in2 := 100.0, out => "DATOS ESCRITURA VFDS"."096P001F".FRECUENCIA)
   END_RUNG
   // the same network as SCL:
   IF "SELEC TAB MODO REMOTO BOMBA 096P001F" AND "MODO OPERACION"."096P001F".MANUAL THEN
       #SA6 := "ESC HZ"."096P001F"."FRECUENCIA OP";
   END_IF;
   IF "MODO OPERACION"."096P001F".SCADA THEN
       #"CONSIGNA 6" := INT_TO_REAL("DATA MODBUS TCP".DATA[98]);
       #SA6 := #"CONSIGNA 6" / 100.0;
   END_IF;
   IF "SELEC TAB MODO REMOTO BOMBA 096P001F" AND "MODO OPERACION"."096P001F".AUTOMATICO THEN
       #SA6 := ((("CONFIG SIS PRESION AGUA SERVICIO"."FRECUENCIA MAXIMA CONFIGURADA EN VFDS"-"CONFIG SIS PRESION AGUA SERVICIO"."FRECUENCIA MINIMA CONFIGURADA EN VFDS")/(100.0-0.0))*"CONSIGNA FRECUENCIA AGUA RESIDUAL")+("CONFIG SIS PRESION AGUA SERVICIO"."FRECUENCIA MINIMA CONFIGURADA EN VFDS"-((("CONFIG SIS PRESION AGUA SERVICIO"."FRECUENCIA MAXIMA CONFIGURADA EN VFDS"-"CONFIG SIS PRESION AGUA SERVICIO"."FRECUENCIA MINIMA CONFIGURADA EN VFDS")/(100.0-0.0))*0.0));
   END_IF;
   IF NOT "SELEC TAB MODO REMOTO BOMBA 096P001F" THEN #SA6 := "ESC HZ"."096P001F"."FRECUENCIA OP"; END_IF;
   "DATOS LECTURA VFDS"."096P001F"."FRECUENCIA %" := (((60.0-0.0)/(60.0-0.0))*"DATOS LECTURA VFDS"."096P001F".FRECUENCIA)+(0.0-(((60.0-0.0)/(60.0-0.0))*0.0));
   "DATOS ESCRITURA VFDS"."096P001F".FRECUENCIA := #SA6 * 100.0;
END_REGION
END_FUNCTION

ORGANIZATION_BLOCK "Main"   // OB1, LAD, ProgramCycle
TITLE = "Main Program Sweep (Cycle)"
{ S7_Optimized_Access := 'TRUE' }
VERSION : 0.1
   VAR_INPUT
      Initial_Call : Bool;   // Initial call of this OB
      Remanence : Bool;   // =True, if remanent data are available
   END_VAR
   VAR_TEMP   // added for the SCL form of the ladder/FBD networks
      _w1 : Bool;
      _w2 : Bool;
   END_VAR
BEGIN

REGION Network 1
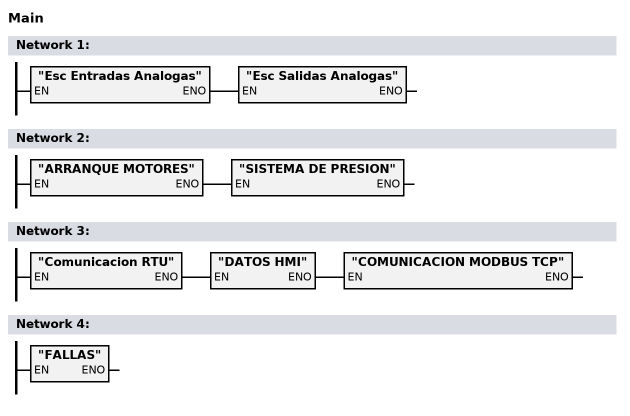
   RUNG wire#powerrail
      "Esc Entradas Analogas"()
      "Esc Salidas Analogas"()
   END_RUNG
   // the same network as SCL:
   "Esc Entradas Analogas"(ENO => #_w1);
   IF #_w1 THEN "Esc Salidas Analogas"(); END_IF;
END_REGION

REGION Network 2
   RUNG wire#powerrail
      "ARRANQUE MOTORES"()
      "SISTEMA DE PRESION"()
   END_RUNG
   // the same network as SCL:
   "ARRANQUE MOTORES"(ENO => #_w1);
   IF #_w1 THEN "SISTEMA DE PRESION"(); END_IF;
END_REGION

REGION Network 3
   RUNG wire#powerrail
      "Comunicacion RTU"()
      "DATOS HMI"()
      "COMUNICACION MODBUS TCP"()
   END_RUNG
   // the same network as SCL:
   "Comunicacion RTU"(ENO => #_w1);
   "DATOS HMI"(EN := #_w1, ENO => #_w2);
   IF #_w2 THEN "COMUNICACION MODBUS TCP"(); END_IF;
END_REGION

REGION Network 4
   RUNG wire#powerrail
      "FALLAS"()
   END_RUNG
   // the same network as SCL:
   "FALLAS"();
END_REGION
END_ORGANIZATION_BLOCK

ORGANIZATION_BLOCK "PIDS"   // OB30, LAD, CyclicInterrupt
{ S7_Optimized_Access := 'TRUE' }
VERSION : 0.1
   VAR_INPUT
      Initial_Call : Bool;   // Initial call of this OB
      Event_Count : Int;   // Events discarded
   END_VAR
   VAR_TEMP
      SETPOINT : Real;
      SETPOINT2 : Real;
   END_VAR
BEGIN

REGION Network 1
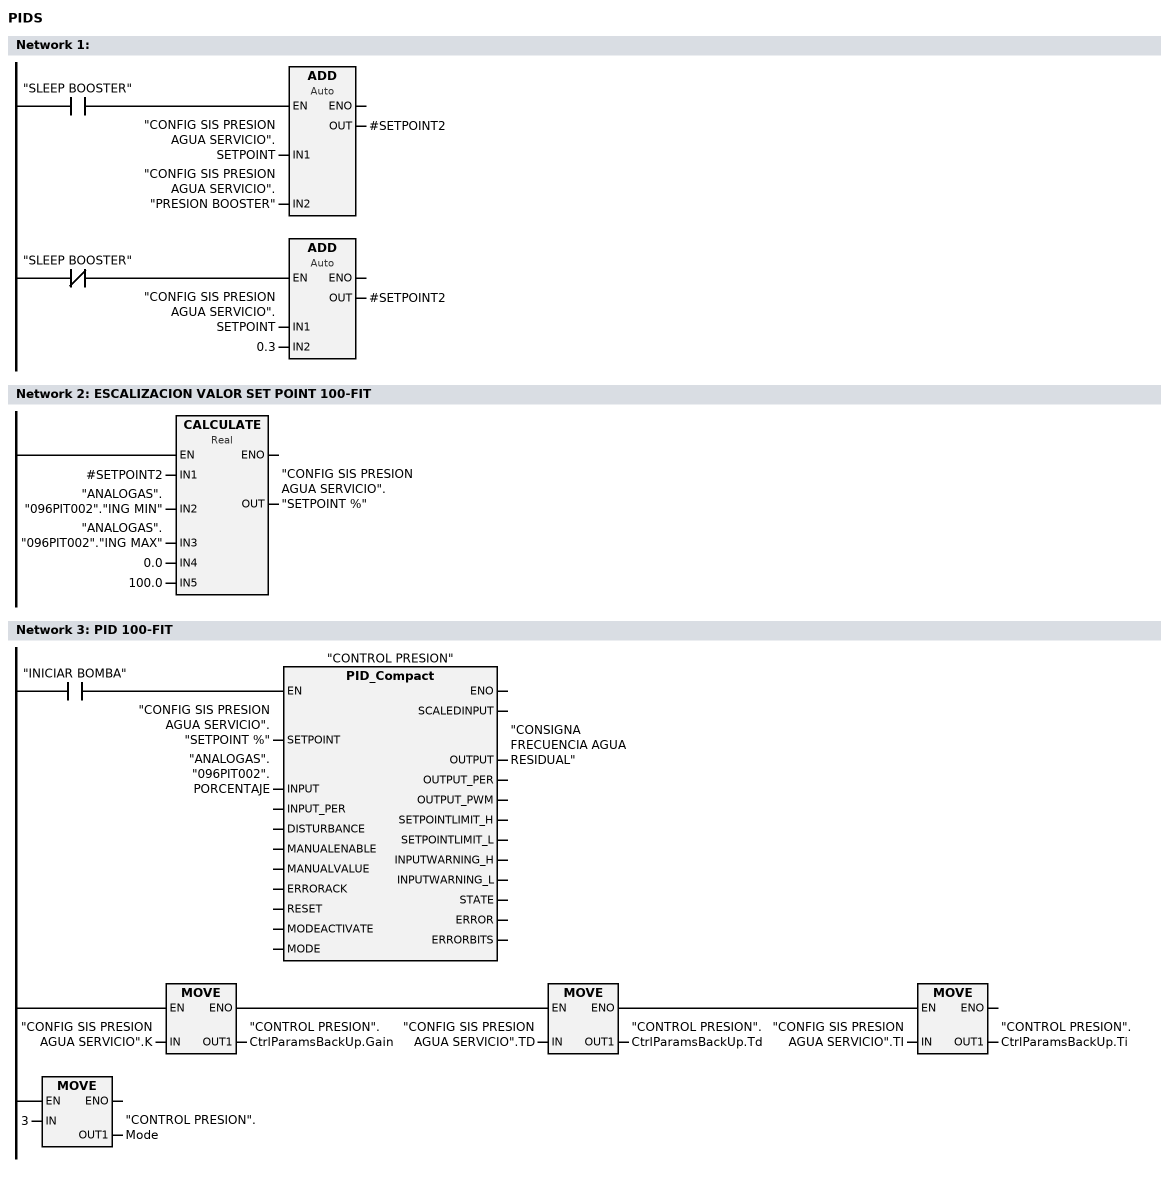
   RUNG wire#powerrail
      Contact( "SLEEP BOOSTER" )
      Add(in1 := "CONFIG SIS PRESION AGUA SERVICIO".SETPOINT, in2 := "CONFIG SIS PRESION AGUA SERVICIO"."PRESION BOOSTER", out => #SETPOINT2)
   END_RUNG
   RUNG wire#powerrail
      I_Contact( "SLEEP BOOSTER" )
      Add(in1 := "CONFIG SIS PRESION AGUA SERVICIO".SETPOINT, in2 := 0.3, out => #SETPOINT2)
   END_RUNG
   // the same network as SCL:
   IF "SLEEP BOOSTER" THEN
       #SETPOINT2 := "CONFIG SIS PRESION AGUA SERVICIO".SETPOINT + "CONFIG SIS PRESION AGUA SERVICIO"."PRESION BOOSTER";
   END_IF;
   IF NOT "SLEEP BOOSTER" THEN #SETPOINT2 := "CONFIG SIS PRESION AGUA SERVICIO".SETPOINT + 0.3; END_IF;
END_REGION

REGION Network 2: ESCALIZACION VALOR SET POINT 100-FIT
   RUNG wire#powerrail
      { S7_Templates := "SrcType := Real"; S7_Expression := "(((IN5-IN4)/(IN3-IN2))*IN1)+(IN4-((IN5-IN4)/(IN3-IN2)*IN2))" } Calculate(in1 := #SETPOINT2, in2 := "ANALOGAS"."096PIT002"."ING MIN", in3 := "ANALOGAS"."096PIT002"."ING MAX", in4 := 0.0, in5 := 100.0, out => "CONFIG SIS PRESION AGUA SERVICIO"."SETPOINT %")
   END_RUNG
   // the same network as SCL:
   "CONFIG SIS PRESION AGUA SERVICIO"."SETPOINT %" := (((100.0-0.0)/("ANALOGAS"."096PIT002"."ING MAX"-"ANALOGAS"."096PIT002"."ING MIN"))*#SETPOINT2)+(0.0-((100.0-0.0)/("ANALOGAS"."096PIT002"."ING MAX"-"ANALOGAS"."096PIT002"."ING MIN")*"ANALOGAS"."096PIT002"."ING MIN"));
END_REGION

REGION Network 3: PID 100-FIT
   IF "INICIAR BOMBA" THEN
       "CONTROL PRESION"(Setpoint := "CONFIG SIS PRESION AGUA SERVICIO"."SETPOINT %",   // PID_Compact
                         Input := "ANALOGAS"."096PIT002".PORCENTAJE,
                         Output => "CONSIGNA FRECUENCIA AGUA RESIDUAL");
   END_IF;
   "CONTROL PRESION".CtrlParamsBackUp.Gain := "CONFIG SIS PRESION AGUA SERVICIO".K;
   "CONTROL PRESION".CtrlParamsBackUp.Td := "CONFIG SIS PRESION AGUA SERVICIO".TD;
   "CONTROL PRESION".CtrlParamsBackUp.Ti := "CONFIG SIS PRESION AGUA SERVICIO".TI;
   "CONTROL PRESION".Mode := 3;
END_REGION
END_ORGANIZATION_BLOCK

// ===== PLC "PLC_2 Compresores y agua potable"  CPU 1214C AC/DC/Rly =====

VAR_GLOBAL   // PLC tag table "Tabla de variables estándar"
   "PARO EMERGENCIA TAB AGUA POTABLE LOCAL" AT %I0.0 : Bool;
   "FALLA GUARDAMOTOR COMPRESOR 096P005A" AT %I0.1 : Bool;
   "FALLA GUARDAMOTOR COMPRESOR 096P005B" AT %I0.2 : Bool;
   "FALLA ARRANCADOR SUAVE COMPRESOR 096P005A" AT %I0.3 : Bool;
   "FALLA ARRANCADOR SUAVE COMPRESOR 096P005B" AT %I0.4 : Bool;
   "SELEC TAB MODO CCM COMPRESOR 096P005A" AT %I0.5 : Bool;
   "SELEC TAB MODO CAMPO COMPRESOR 096P005A" AT %I0.6 : Bool;
   "SELEC TAB MODO REMOTO COMPRESOR 096P005A" AT %I0.7 : Bool;
   "SELEC TAB MODO CCM COMPRESOR 096P005B" AT %I1.0 : Bool;
   "SELEC TAB MODO CAMPO COMPRESOR 096P005B" AT %I1.1 : Bool;
   "SELEC TAB MODO REMOTO COMPRESOR 096P005B" AT %I1.2 : Bool;
   "SELEC TAB MODO CCM BOMBA 096P004A" AT %I1.3 : Bool;
   "SELEC TAB MODO CAMPO BOMBA 096P004A" AT %I1.4 : Bool;
   "SELEC TAB MODO REMOTO BOMBA 096P004A" AT %I1.5 : Bool;
   "SELEC TAB MODO CCM BOMBA 096P004B" AT %I2.0 : Bool;
   "SELEC TAB MODO CAMPO BOMBA 096P004B" AT %I2.1 : Bool;
   "SELEC TAB MODO REMOTO BOMBA 096P004B" AT %I2.2 : Bool;
   "SELEC TAB MODO CCM BOMBA 096P004C" AT %I2.3 : Bool;
   "SELEC TAB MODO CAMPO BOMBA 096P004C" AT %I2.4 : Bool;
   "SELEC TAB MODO REMOTO BOMBA 096P004C" AT %I2.5 : Bool;
   "SELEC TAB MODO CCM BOMBA 096P004D" AT %I2.6 : Bool;
   "SELEC TAB MODO CAMPO BOMBA 096P004D" AT %I2.7 : Bool;
   "SELEC TAB MODO REMOTO BOMBA 096P004D" AT %I3.0 : Bool;
   "PULSADOR START CCM 096P005A" AT %I3.1 : Bool;
   "PULSADOR STOP CCM 096P005A" AT %I3.2 : Bool;
   "PULSADOR START CCM 096P005B" AT %I3.3 : Bool;
   "PULSADOR STOP CCM 096P005B" AT %I3.4 : Bool;
   "PULSADOR START CCM 096P004A" AT %I3.5 : Bool;
   "PULSADOR STOP CCM 096P004A" AT %I3.6 : Bool;
   "PULSADOR START CCM 096P004B" AT %I3.7 : Bool;
   "PULSADOR STOP CCM 096P004B" AT %I4.0 : Bool;
   "PULSADOR START CCM 096P004C" AT %I4.1 : Bool;
   "PULSADOR STOP CCM 096P004C" AT %I4.2 : Bool;
   "PULSADOR START CCM 096P004D" AT %I4.3 : Bool;
   "PULSADOR STOP CCM 096P004D" AT %I4.4 : Bool;
   "PULSADOR RESET CCM 096P005A" AT %I4.5 : Bool;
   "PULSADOR RESET CCM 096P005B" AT %I4.6 : Bool;
   "PULSADOR RESET CCM 096P004A" AT %I4.7 : Bool;
   "PULSADOR RESET CCM 096P004B" AT %I5.0 : Bool;
   "PULSADOR RESET CCM 096P004C" AT %I5.1 : Bool;
   "PULSADOR RESET CCM 096P004D" AT %I5.2 : Bool;
   "PARO EMERGENCIA BOMBAS 096P005A" AT %I5.3 : Bool;
   "PULSADOR START CAMPO 096P005A" AT %I5.4 : Bool;
   "PULSADOR STOP CAMPO 096P005A" AT %I5.5 : Bool;
   "PULSADOR START CAMPO 096P005B" AT %I5.6 : Bool;
   "PULSADOR STOP CAMPO 096P005B" AT %I5.7 : Bool;
   "PULSADOR START CAMPO 096P004A" AT %I6.1 : Bool;
   "PULSADOR STOP CAMPO 096P004A" AT %I6.2 : Bool;
   "PULSADOR START CAMPO 096P004B" AT %I6.3 : Bool;
   "PULSADOR STOP CAMPO 096P004B" AT %I6.4 : Bool;
   "PULSADOR START CAMPO 096P004C" AT %I6.5 : Bool;
   "PULSADOR STOP CAMPO 096P004C" AT %I6.6 : Bool;
   "PULSADOR START CAMPO 096P004D" AT %I6.7 : Bool;
   "PULSADOR STOP CAMPO 096P004D" AT %I7.0 : Bool;
   "PARO EMERGENCIA BOMBAS 096P005B" AT %I6.0 : Bool;
   "SWITCH DE BAJA PRESION 096P005A" AT %I8.1 : Bool;
   "SWITCH DE FLUJO 096P005A" AT %I8.2 : Bool;
   "SWITCH DE BAJA PRESION 096P005B" AT %I8.3 : Bool;
   "SWITCH DE FLUJO 096P005B" AT %I8.4 : Bool;
   "SWITCH DE BAJA PRESION AGUA POTABLE" AT %I8.5 : Bool;
   "SWITCH DE FLUJO AGUA POTABLE" AT %I8.6 : Bool;
   "TRANSMISOR PRESION SUCCION BOMBA 096PIT005" AT %IW300 : Word;
   "TRANSMISOR PRESION DESCARGA BOMBA 096PIT008" AT %IW302 : Word;
   "TRANSMISOR PRESION SUCCION BOMBA 096PIT009" AT %IW304 : Word;
   "TRANSMISOR PRESION DESCARGA BOMBA 096PIT010" AT %IW306 : Word;
   "TRANSMISOR PRESION SUCCION BOMBA 096PIT004" AT %IW308 : Word;
   "TRANSMISOR PRESION DESCARGA BOMBA 096PIT006" AT %IW310 : Word;
   "PARO EMERGENCIA BOMBAS 096P004A" AT %I8.7 : Bool;
   "PARO EMERGENCIA BOMBAS 096P004B" AT %I9.0 : Bool;
   "PARO EMERGENCIA BOMBAS 096P004C" AT %I9.1 : Bool;
   "PARO EMERGENCIA BOMBAS 096P004D" AT %I9.2 : Bool;
   "PERMISO DE ARRANQUE BIOGAS 1" AT %I9.3 : Bool;
   "PERMISO DE ARRANQUE POTABLE 1" AT %I9.4 : Bool;
   "PERMISO DE ARRANQUE POTABLE 2" AT %I9.5 : Bool;
   "PERMISO DE ARRANQUE BIOGAS 2" AT %I9.6 : Bool;
   "OPERANDO BOMBA 096P005A" AT %Q0.0 : Bool;
   "FALLA BOMBA 096P005A" AT %Q0.1 : Bool;
   "OPERANDO BOMBA 096P005B" AT %Q0.2 : Bool;
   "FALLA BOMBA 096P005B" AT %Q0.3 : Bool;
   "OPERANDO BOMBA 096P004A" AT %Q0.4 : Bool;
   "FALLA BOMBA 096P004A" AT %Q0.5 : Bool;
   "OPERANDO BOMBA 096P004B" AT %Q0.6 : Bool;
   "FALLA BOMBA 096P004B" AT %Q0.7 : Bool;
   "OPERANDO BOMBA 096P004C" AT %Q1.0 : Bool;
   "FALLA BOMBA 096P004C" AT %Q1.1 : Bool;
   "OPERANDO BOMBA 096P004D" AT %Q2.0 : Bool;
   "FALLA BOMBA 096P004D" AT %Q2.1 : Bool;
   "HABILITACION SISTEMA 5A" AT %M0.0 : Bool;
   "HABILITACION SISTEMA 5B" AT %M0.1 : Bool;
   "BOMBA LIDER BIOGAS 1" AT %M0.2 : Bool;
   "BOMBA LIDER BIOGAS 2" AT %M0.3 : Bool;
   "DISPONIBLE BOMBA 5A" AT %M0.4 : Bool;
   "DISPONIBLE BOMBA 5B" AT %M0.5 : Bool;
   "INICIAR BOMBA BIOGAS 1" AT %M0.6 : Bool;
   "INICIAR BOMBA BIOGAS 2" AT %M0.7 : Bool;
   "System_Byte" AT %MB200 : Byte;
   "FirstScan" AT %M200.0 : Bool;
   "DiagStatusUpdate" AT %M200.1 : Bool;
   "AlwaysTRUE" AT %M200.2 : Bool;
   "AlwaysFALSE" AT %M200.3 : Bool;
   "Clock_Byte" AT %MB201 : Byte;
   "Clock_10Hz" AT %M201.0 : Bool;
   "Clock_5Hz" AT %M201.1 : Bool;
   "Clock_2.5Hz" AT %M201.2 : Bool;
   "Clock_2Hz" AT %M201.3 : Bool;
   "Clock_1.25Hz" AT %M201.4 : Bool;
   "Clock_1Hz" AT %M201.5 : Bool;
   "Clock_0.625Hz" AT %M201.6 : Bool;
   "Clock_0.5Hz" AT %M201.7 : Bool;
   "Tag_4" AT %M10.0 : Bool;
   "Tag_5" AT %M10.1 : Bool;
   "Tag_6" AT %M10.2 : Bool;
   "Tag_7" AT %M10.3 : Bool;
   "Tag_2" AT %M1.0 : Bool;
   "Tag_15" AT %M1.1 : Bool;
   "Tag_16" AT %M1.2 : Bool;
   "Tag_1" AT %M1.3 : Bool;
   "Tag_3" AT %M1.4 : Bool;
   "Tag_8" AT %M1.5 : Bool;
   "Tag_9" AT %M1.6 : Bool;
   "Tag_10" AT %M1.7 : Bool;
   "Tag_11" AT %M2.0 : Bool;
   "Tag_12" AT %M2.1 : Bool;
   "Tag_13" AT %M2.2 : Bool;
   "Tag_14" AT %M2.3 : Bool;
   "Tag_17" AT %M2.4 : Bool;
   "Tag_18" AT %M2.5 : Bool;
   "Tag_19" AT %M2.6 : Bool;
   "Tag_20" AT %M2.7 : Bool;
   "Tag_21" AT %M3.0 : Bool;
   "Tag_22" AT %M3.1 : Bool;
   "HABILITACION SISTEMA" AT %M3.2 : Bool;
   "INICIAR BOMBA" AT %M3.3 : Bool;
   "BOMBA LIDER 1" AT %M3.4 : Bool;
   "ARRANQUE BOMBA A" AT %M3.5 : Bool;
   "BOMBA LIDER 2" AT %M3.6 : Bool;
   "ARRANQUE BOMBA B" AT %M3.7 : Bool;
   "BOMBA LIDER 3" AT %M4.0 : Bool;
   "ARRANQUE BOMBA C" AT %M4.1 : Bool;
   "BOMBA LIDER 4" AT %M4.2 : Bool;
   "ARRANQUE BOMBA D" AT %M4.3 : Bool;
   "DISPONIBLE BOMBA A" AT %M4.4 : Bool;
   "DISPONIBLE BOMBA B" AT %M4.5 : Bool;
   "DISPONIBLE BOMBA C" AT %M4.6 : Bool;
   "DISPONIBLE BOMBA D" AT %M4.7 : Bool;
   "SLEEP BOOSTER" AT %M5.0 : Bool;
   "CONSIGNA FRECUENCIA AGUA RESIDUAL" AT %MD100 : Real;
   "PRESION OK" AT %M5.1 : Bool;
   "AD1" AT %M5.2 : Bool;
   "AD2" AT %M5.3 : Bool;
   "AD3" AT %M5.4 : Bool;
   "Tag_23" AT %M11.0 : Bool;
   "Tag_24" AT %M11.1 : Bool;
   "Tag_25" AT %M11.2 : Bool;
   "Tag_26" AT %M11.3 : Bool;
   "Tag_27" AT %M11.4 : Bool;
   "Tag_28" AT %M11.5 : Bool;
   "Tag_29" AT %M11.6 : Bool;
   "Tag_30" AT %M11.7 : Bool;
   "Tag_31" AT %M80.0 : Bool;
   "Tag_32" AT %M30.0 : Bool;
   "Tag_33" AT %M40.0 : Bool;
   "Tag_34" AT %M40.1 : Bool;
   "Tag_35" AT %M40.2 : Bool;
   "Tag_36" AT %M40.3 : Bool;
END_VAR

TYPE "typeSoftStarterDiagnostics"
VERSION : 0.1
   STRUCT
      ready : Bool;
      motorRight : Bool;
      motorLeft : Bool;
      switchingElementOverload : Bool;
      switchingElementDefective : Bool;
      emergencyStartActive : Bool;
      groupError : Bool;
      groupWarning : Bool;
      reserve_33800 : Bool;
      noMainPower : Bool;
      reserve_33802 : Bool;
      startModeActive : Bool;
      stopModeActive : Bool;
      reserve_33805 : Bool;
      electricalBrakingActive : Bool;
      creepSpeedActive : Bool;
      temperatureSensorOverload : Bool;
      temperatureSensorWireBreak : Bool;
      temperatureSensorShortCircuit : Bool;
      thermalMotorModelOverload : Bool;
      mototrOverloadShutoff : Bool;
      idleTimeActive : Bool;
      coolingTimeActive : Bool;
      reserve_33815 : Bool;
      reserve_33816 : Bool;
      reserve_33817 : Bool;
      reserve_33818 : Bool;
      currentLimitingActive : Bool;
      reserve_33820 : Bool;
      reserve_33821 : Bool;
      generatorOperation : Bool;
      inputControl : Bool;
      asymmetryLimitErrorExceeded : Bool;
      asymmetryShutoff : Bool;
      currentLimitErrorExceeded : Bool;
      currentLimitErrorUndershot : Bool;
      currentErrorLimitShutoff : Bool;
      reserve_33829 : Bool;
      reserve_33830 : Bool;
      reserve_33831 : Bool;
      input1 : Bool;
      input2 : Bool;
      input3 : Bool;
      input4 : Bool;
      reserve_33836 : Bool;
      reserve_33837 : Bool;
      reserve_33838 : Bool;
      reserve_33839 : Bool;
      groundFaultLimitErrorExceeded : Bool;
      reserve_33841 : Bool;
      quickStopActive : Bool;
      reserve_33843 : Bool;
      reserve_33844 : Bool;
      reserve_33845 : Bool;
      maximumPointerReset : Bool;
      electronicsSupplyVoltageTooLow : Bool;
      busError : Bool;
      masterCpuStop : Bool;
      automaticMode : Bool;
      operatingModeManual : Bool;
      manualOperationLocal : Bool;
      reserve_33853 : Bool;
      connectionAbortInManualMode : Bool;
      processImageError : Bool;
      parameterAssignmentActive : Bool;
      invalidParameter : Bool;
      parametersCannotBeChangedInONState : Bool;
      parametersDisableCpuMasterActive : Bool;
      noExternalStartParametersReceived : Bool;
      reserve_33861 : Bool;
      reserve_33862 : Bool;
      reserve_33863 : Bool;
      selfTestActive : Bool;
      reserve_33865 : Bool;
      errorDuringSelfTest : Bool;
      factorySettingRestored : Bool;
      reserve_33868 : Bool;
      reserve_33869 : Bool;
      reserve_33870 : Bool;
      reserve_33871 : Bool;
      parameterNumberError : UInt;
      reserve_33888 : Bool;
      reserve_33889 : Bool;
      reserve_33890 : Bool;
      presetUnequalActualConfiguration : Bool;
      reserve_33892 : Bool;
      temperatureSensorOverload_1 : Bool;
      temperatureSensorWireBreak_1 : Bool;
      temperatureSensorShortCircuit_1 : Bool;
      parameterSet1Active : Bool;
      parameterSet2Active : Bool;
      parameterSet3Active : Bool;
      reserve_33899 : Bool;
      parameterSetChangeNotPossible : Bool;
      reserve_33901 : Bool;
      presetUnequalActualConfiguration_1 : Bool;
      typeOfMotorConnectionWrong : Bool;
      reserve_33904 : Bool;
      reserve_33905 : Bool;
      motorHeatingActive : Bool;
      dcBrakingActive : Bool;
      dynamicDCBrakingActive : Bool;
      typeOfMotorConnectionStandard : Bool;
      typeOfMotorConnectionInsideDelta : Bool;
      motorConnectionTypeUnknown : Bool;
      loadMissing : Bool;
      reserve_33913 : Bool;
      phaseFailureL1 : Bool;
      phaseFailureL2 : Bool;
      phaseFailureL3 : Bool;
      mainPowerRotationRight : Bool;
      mainPowerRotationLeft : Bool;
      reserve_33919 : Bool;
      reserve_33920 : Bool;
      reserve_33921 : Bool;
      reserve_33922 : Bool;
      reserve_33923 : Bool;
      reserve_33924 : Bool;
      reserve_33925 : Bool;
      reserve_33926 : Bool;
      reserve_33927 : Bool;
      output1Active : Bool;
      output2Active : Bool;
      output3Active : Bool;
      output4Active : Bool;
      output1TimeActive : Bool;
      output2TimeActive : Bool;
      reserve_33934 : Bool;
      output4TimeActive : Bool;
      reserve_33936 : Bool;
      reserve_33937 : Bool;
      reserve_33938 : Bool;
      reserve_33939 : Bool;
      reserve_33940 : Bool;
      reserve_33941 : Bool;
      reserve_33942 : Bool;
      reserve_33943 : Bool;
      reserve_33944 : Bool;
      readyToStartForMotorOn : Bool;
      reserve_33946 : Bool;
      bypassDefective : Bool;
      bypassProtectiveShutoff : Bool;
      switchingElementL1Defective : Bool;
      switchingElementL2Defective : Bool;
      switchingElementL3Defective : Bool;
      thermalMotorModelDeactivated : Bool;
      reserve_33953 : Bool;
      reserve_33954 : Bool;
      phaseAngleControlFailure : Bool;
      reserve_33956 : Bool;
      reserve_33957 : Bool;
      reserve_33958 : Bool;
      reserve_33959 : Bool;
      switchingElementCoolingTimeActive : Bool;
      switchingElementForStartTooHot : Bool;
      currentMeasuringRangeOvershot : Bool;
      reserve_33963 : Bool;
      reserve_33964 : Bool;
      reserve_33965 : Bool;
      reserve_33966 : Bool;
      reserve_33967 : Bool;
      automaticMode_1 : Bool;
      operatingModeManual_1 : Bool;
      manualOperationBusPcControlled : Bool;
      manualOperationLocal_1 : Bool;
      manualOperationLocalInputControlled : Bool;
      manualOperationLocalHmiControlled : Bool;
      manualOperationLocalPcControlled : Bool;
      reserve_33975 : Bool;
      reserve_33976 : Bool;
      reserve_33977 : Bool;
      reserve_33978 : Bool;
      reserve_33979 : Bool;
      reserve_33980 : Bool;
      reserve_33981 : Bool;
      reserve_33982 : Bool;
      reserve_33983 : Bool;
      reserve_33984 : Bool;
      reserve_33985 : Bool;
      reserve_33986 : Bool;
      reserve_33987 : Bool;
      reserve_33988 : Bool;
      reserve_33989 : Bool;
      reserve_33990 : Bool;
      reserve_33991 : Bool;
      deviceError : Bool;
      reserve_33993 : Bool;
      reserve_33994 : Bool;
      reserve_33995 : Bool;
      reserve_33996 : Bool;
      reserve_33997 : Bool;
      reserve_33998 : Bool;
      reserve_33999 : Bool;
      reserve_34000 : Bool;
      reserve_34001 : Bool;
      reserve_34002 : Bool;
      reserve_34003 : Bool;
      reserve_34004 : Bool;
      reserve_34005 : Bool;
      reserve_34006 : Bool;
      reserve_34007 : Bool;
      reserve_34008 : Bool;
      reserve_34009 : Bool;
      reserve_34010 : Bool;
      reserve_34011 : Bool;
      reserve_34012 : Bool;
      reserve_34013 : Bool;
      reserve_34014 : Bool;
      reserve_34015 : Bool;
      updateFirmwareRejected : Bool;
      updateFirmwareActive : Bool;
      updateFirmwareSuccessful : Bool;
      updateFirmwareUnsuccessful : Bool;
      reserve_34020 : Bool;
      reserve_34021 : Bool;
      reserve_34022 : Bool;
      reserve_34023 : Bool;
      reserve_34024 : Bool;
      reserve_34025 : Bool;
      reserve_34026 : Bool;
      reserve_34027 : Bool;
      reserve_34028 : Bool;
      reserve_34029 : Bool;
      reserve_34030 : Bool;
      operationBypassActive : Bool;
      reserve_34032 : Bool;
      reserve_34033 : Bool;
      reserve_34034 : Bool;
      reserve_34035 : Bool;
      reserve_34036 : Bool;
      reserve_34037 : Bool;
      reserve_34038 : Bool;
      reserve_34039 : Bool;
      reserve_34040 : Bool;
      reserve_34041 : Bool;
      reserve_34042 : Bool;
      reserve_34043 : Bool;
      reserve_34044 : Bool;
      reserve_34045 : Bool;
      reserve_34046 : Bool;
      reserve_34047 : Bool;
      reserve_34048 : Bool;
      reserve_34049 : Bool;
      reserve_34050 : Bool;
      reserve_34051 : Bool;
      reserve_34052 : Bool;
      reserve_34053 : Bool;
      reserve_34054 : Bool;
      reserve_34055 : Bool;
      reserve_34056 : Bool;
      reserve_34057 : Bool;
      reserve_34058 : Bool;
      reserve_34059 : Bool;
      reserve_34060 : Bool;
      reserve_34061 : Bool;
      reserve_34062 : Bool;
      reserve_34063 : Bool;
      reserve_34064 : Bool;
      reserve_34065 : Bool;
      reserve_34066 : Bool;
      reserve_34067 : Bool;
      reserve_34068 : Bool;
      reserve_34069 : Bool;
      reserve_34070 : Bool;
      reserve_34071 : Bool;
      reserve_34072 : Bool;
      reserve_34073 : Bool;
      reserve_34074 : Bool;
      reserve_34075 : Bool;
      reserve_34076 : Bool;
      reserve_34077 : Bool;
      reserve_34078 : Bool;
      reserve_34079 : Bool;
      reserve_34080 : Bool;
      reserve_34081 : Bool;
      reserve_34082 : Bool;
      reserve_34083 : Bool;
      reserve_34084 : Bool;
      reserve_34085 : Bool;
      reserve_34086 : Bool;
      reserve_34087 : Bool;
      reserve_34088 : Bool;
      reserve_34089 : Bool;
      reserve_34090 : Bool;
      reserve_34091 : Bool;
      reserve_34092 : Bool;
      reserve_34093 : Bool;
      reserve_34094 : Bool;
      reserve_34095 : Bool;
      reserve_34096 : Bool;
      reserve_34097 : Bool;
      reserve_34098 : Bool;
      reserve_34099 : Bool;
      reserve_34100 : Bool;
      reserve_34101 : Bool;
      reserve_34102 : Bool;
      reserve_34103 : Bool;
      reserve_34104 : Bool;
      reserve_34105 : Bool;
      reserve_34106 : Bool;
      reserve_34107 : Bool;
      reserve_34108 : Bool;
      reserve_34109 : Bool;
      reserve_34110 : Bool;
      reserve_34111 : Bool;
      reserve_34112 : Bool;
      reserve_34113 : Bool;
      reserve_34114 : Bool;
      reserve_34115 : Bool;
      reserve_34116 : Bool;
      reserve_34117 : Bool;
      reserve_34118 : Bool;
      reserve_34119 : Bool;
      reserve_34120 : Bool;
      reserve_34121 : Bool;
      reserve_34122 : Bool;
      reserve_34123 : Bool;
      reserve_34124 : Bool;
      reserve_34125 : Bool;
      reserve_34126 : Bool;
      reserve_34127 : Bool;
      reserve_34128 : Bool;
      reserve_34129 : Bool;
      reserve_34130 : Bool;
      reserve_34131 : Bool;
      reserve_34132 : Bool;
      reserve_34133 : Bool;
      normalOperationActive : Bool;
      reserve_34135 : Bool;
      reserve_34136 : Bool;
      reserve_34137 : Bool;
      reserve_34138 : Bool;
      testOperationActive : Bool;
      reserve_34140 : Bool;
      reserve_34141 : Bool;
      reserve_34142 : Bool;
      reserve_34143 : Bool;
      reserve_34144 : Bool;
      reserve_34145 : Bool;
      reserve_34146 : Bool;
      reserve_34147 : Bool;
      reserve_34148 : Bool;
      reserve_34149 : Bool;
      reserve_34150 : Bool;
      reserve_34151 : Bool;
      reserve_34152 : Bool;
      reserve_34153 : Bool;
      reserve_34154 : Bool;
      reserve_34155 : Bool;
      reserve_34156 : Bool;
      reserve_34157 : Bool;
      reserve_34158 : Bool;
      reserve_34159 : Bool;
      reserve_34160 : Bool;
      reserve_34161 : Bool;
      reserve_34162 : Bool;
      reserve_34163 : Bool;
      reserve_34164 : Bool;
      reserve_34165 : Bool;
      reserve_34166 : Bool;
      reserve_34167 : Bool;
      reserve_34168 : Bool;
      reserve_34169 : Bool;
      reserve_34170 : Bool;
      reserve_34171 : Bool;
      reserve_34172 : Bool;
      reserve_34173 : Bool;
      reserve_34174 : Bool;
      reserve_34175 : Bool;
      reserve_34176 : Bool;
      reserve_34177 : Bool;
      reserve_34178 : Bool;
      reserve_34179 : Bool;
      reserve_34180 : Bool;
      reserve_34181 : Bool;
      reserve_34182 : Bool;
      reserve_34183 : Bool;
      reserve_34184 : Bool;
      reserve_34185 : Bool;
      reserve_34186 : Bool;
      reserve_34187 : Bool;
      reserve_34188 : Bool;
      reserve_34189 : Bool;
      reserve_34190 : Bool;
      reserve_34191 : Bool;
      EXApplicationActive : Bool;
      reserve_34193 : Bool;
      NewExParameterValuesDetected : Bool;
      reserve_34195 : Bool;
      reserve_34196 : Bool;
      releaseDeniedDueToWrongFParameterCRC : Bool;
      reserve_34198 : Bool;
      reserve_34199 : Bool;
      reserve_34200 : Bool;
      reserve_34201 : Bool;
      reserve_34202 : Bool;
      reserve_34203 : Bool;
      reserve_34204 : Bool;
      reserve_34205 : Bool;
      reserve_34206 : Bool;
      reserve_34207 : Bool;
      reserve_34208 : Bool;
      reserve_34209 : Bool;
      remainingTimeForTrippingWarningLimitUndershot : Bool;
      motorHeatingWarningLimitExceeded : Bool;
      currentLimitMaintenanceDemandedExceeded : Bool;
      currentLimitMaintenanceDemandedUndershot : Bool;
      asymmetryLimitWarningExceeded : Bool;
      groundFaultLimitWarningExceeded : Bool;
      reserve_34216 : Bool;
      reserve_34217 : Bool;
      reserve_34218 : Bool;
      reserve_34219 : Bool;
      reserve_34220 : Bool;
      reserve_34221 : Bool;
      reserve_34222 : Bool;
      reserve_34223 : Bool;
      reserve_34224 : Bool;
      reserve_34225 : Bool;
      reserve_34226 : Bool;
      reserve_34227 : Bool;
      reserve_34228 : Bool;
      reserve_34229 : Bool;
      reserve_34230 : Bool;
      reserve_34231 : Bool;
      pumpCleaningActive : Bool;
      reserve_34233 : Bool;
      reserve_34234 : Bool;
      reserve_34235 : Bool;
      reserve_34236 : Bool;
      reserve_34237 : Bool;
      reserve_34238 : Bool;
      reserve_34239 : Bool;
      reserve_34240 : Bool;
      reserve_34241 : Bool;
      reserve_34242 : Bool;
      reserve_34243 : Bool;
      reserve_34244 : Bool;
      analogOutputUnderflow : Bool;
      reserve_34246 : Bool;
      reserve_34247 : Bool;
      reserve_34248 : Bool;
      reserve_34249 : Bool;
      reserve_34250 : Bool;
      reserve_34251 : Bool;
      reserve_34252 : Bool;
      analogOutputOverflow : Bool;
      reserve_34254 : Bool;
      reserve_34255 : Bool;
      reserve_34256 : Bool;
      reserve_34257 : Bool;
      reserve_34258 : Bool;
      reserve_34259 : Bool;
      reserve_34260 : Bool;
      reserve_34261 : Bool;
      reserve_34262 : Bool;
      reserve_34263 : Bool;
      reserve_34264 : Bool;
      reserve_34265 : Bool;
      reserve_34266 : Bool;
      reserve_34267 : Bool;
      reserve_34268 : Bool;
      reserve_34269 : Bool;
      reserve_34270 : Bool;
      reserve_34271 : Bool;
      missingInitializationAfterMaintenance : Bool;
      reserve_34273 : Bool;
      reserve_34274 : Bool;
      reserve_34275 : Bool;
      reserve_34276 : Bool;
      reserve_34277 : Bool;
      reserve_34278 : Bool;
      reserve_34279 : Bool;
      switchingFrequencyTimeRunning : Bool;
      switchingFrequencyTimeNotKept : Bool;
      reserve_34282 : Bool;
      switchingFrequencyTimeNotKept_1 : Bool;
      reserve_34284 : Bool;
      reserve_34285 : Bool;
      reserve_34286 : Bool;
      switchingFrequencyLockActive : Bool;
      reserve_34288 : Bool;
      reserve_34289 : Bool;
      emergencyStartEnabled : Bool;
      reserve_34291 : Bool;
      reserve_34292 : Bool;
      reserve_34293 : Bool;
      reserve_34294 : Bool;
      reserve_34295 : Bool;
      reserve_34296 : Bool;
      alternativeStoppingModeActive : Bool;
      reserve_34298 : Bool;
      reserve_34299 : Bool;
      reserve_34300 : Bool;
      reserve_34301 : Bool;
      reserve_34302 : Bool;
      reserve_34303 : Bool;
      reversingDCBrakingActive : Bool;
      reserve_34305 : Bool;
      reserve_34306 : Bool;
      reserve_34307 : Bool;
      reserve_34308 : Bool;
      reserve_34309 : Bool;
      reserve_34310 : Bool;
      reserve_34311 : Bool;
      mainPowerRotationFaulty : Bool;
      reserve_34313 : Bool;
      reserve_34314 : Bool;
      mainPowerRotationFaulty_1 : Bool;
      reserve_34316 : Bool;
      reserve_34317 : Bool;
      reserve_34318 : Bool;
      reserve_34319 : Bool;
      reserve_34320 : Bool;
      reserve_34321 : Bool;
      reserve_34322 : Bool;
      reserve_34323 : Bool;
      reserve_34324 : Bool;
      reserve_34325 : Bool;
      reserve_34326 : Bool;
      reserve_34327 : Bool;
      reserve_34328 : Bool;
      reserve_34329 : Bool;
      reserve_34330 : Bool;
      reserve_34331 : Bool;
      reserve_34332 : Bool;
      checkFan : Bool;
      reserve_34334 : Bool;
      reserve_34335 : Bool;
      reserve_34336 : Bool;
      reserve_34337 : Bool;
      reserve_34338 : Bool;
      reserve_34339 : Bool;
      reserve_34340 : Bool;
      reserve_34341 : Bool;
      reserve_34342 : Bool;
      reserve_34343 : Bool;
      reserve_34344 : Bool;
      reserve_34345 : Bool;
      reserve_34346 : Bool;
      reserve_34347 : Bool;
      reserve_34348 : Bool;
      reserve_34349 : Bool;
      reserve_34350 : Bool;
      reserve_34351 : Bool;
      reserve_34352 : Bool;
      reserve_34353 : Bool;
      reserve_34354 : Bool;
      reserve_34355 : Bool;
      reserve_34356 : Bool;
      reserve_34357 : Bool;
      reserve_34358 : Bool;
      reserve_34359 : Bool;
      reserve_34360 : Bool;
      reserve_34361 : Bool;
      reserve_34362 : Bool;
      reserve_34363 : Bool;
      reserve_34364 : Bool;
      reserve_34365 : Bool;
      reserve_34366 : Bool;
      reserve_34367 : Bool;
      reserve_34368 : Bool;
      reserve_34369 : Bool;
      reserve_34370 : Bool;
      reserve_34371 : Bool;
      reserve_34372 : Bool;
      reserve_34373 : Bool;
      reserve_34374 : Bool;
      reserve_34375 : Bool;
      reserve_34376 : Bool;
      reserve_34377 : Bool;
      activePowerLimitMaintenanceDemandedExceeded : Bool;
      activePowerLimitMaintenanceDemandedUndershot : Bool;
      activePowerErrorLimitExceeded : Bool;
      activePowerErrorLimitUndershot : Bool;
      activePowerErrorLimitShutoff : Bool;
      reserve_34383 : Bool;
      reserve_34384 : Bool;
      reserve_34385 : Bool;
      reserve_34386 : Bool;
      reserve_34387 : Bool;
      reserve_34388 : Bool;
      reserve_34389 : Bool;
      reserve_34390 : Bool;
      reserve_34391 : Bool;
      reserve_34392 : Bool;
      reserve_34393 : Bool;
      reserve_34394 : Bool;
      reserve_34395 : Bool;
      reserve_34396 : Bool;
      reserve_34397 : Bool;
      reserve_34398 : Bool;
      reserve_34399 : Bool;
      reserve_34400 : Bool;
      reserve_34401 : Bool;
      reserve_34402 : Bool;
      reserve_34403 : Bool;
      reserve_34404 : Bool;
      reserve_34405 : Bool;
      reserve_34406 : Bool;
      reserve_34407 : Bool;
      supplyVoltageNotPermittedForTest : Bool;
      supplyVoltageRequiredForTest : Bool;
      reserve_34410 : Bool;
      reserve_34411 : Bool;
      simulationActive : Bool;
      "testWithSmall LoadActive" : Bool;
      reserve_34414 : Bool;
      reserve_34415 : Bool;
      reserve_34416 : Bool;
      reserve_34417 : Bool;
      reserve_34418 : Bool;
      reserve_34419 : Bool;
      reserve_34420 : Bool;
      reserve_34421 : Bool;
      reserve_34422 : Bool;
      reserve_34423 : Bool;
      reserve_34424 : Bool;
      reserve_34425 : Bool;
      reserve_34426 : Bool;
      reserve_34427 : Bool;
      reserve_34428 : Bool;
      reserve_34429 : Bool;
      reserve_34430 : Bool;
      reserve_34431 : Bool;
      operatingTemperatureTooHigh : Bool;
      reserve_34433 : Bool;
      reserve_34434 : Bool;
      reserve_34435 : Bool;
      reserve_34436 : Bool;
      reserve_34437 : Bool;
      reserve_34438 : Bool;
      reserve_34439 : Bool;
      automaticParameterizationActive : Bool;
      reserve_34441 : Bool;
      reserve_34442 : Bool;
      reserve_34443 : Bool;
      reserve_34444 : Bool;
      reserve_34445 : Bool;
      reserve_34446 : Bool;
      reserve_34447 : Bool;
      reserve_34448 : Bool;
      reserve_34449 : Bool;
      startingTimeLimitMaintenanceDemandedExceeded : Bool;
      startingTimeLimitMaintenanceDemandedUndershot : Bool;
      reserve_34452 : Bool;
      reserve_34453 : Bool;
      reserve_34454 : Bool;
      reserve_34455 : Bool;
      logbookApplicationErrorsDeleted : Bool;
      reserve_34457 : Bool;
      logbookApplicationWarningsDeleted : Bool;
      reserve_34459 : Bool;
      logbookApplicationEventDeleted : Bool;
      logbookServiceErrorDeleted : Bool;
      reserve_34462 : Bool;
      logbookServiceEventDeleted : Bool;
   END_STRUCT;
END_TYPE

TYPE "typeMeasuredValues"
VERSION : 0.1
   STRUCT
      reserve_34816 : UInt;
      phaseCurrentL_1 : USInt;
      phaseCurrentL_2 : USInt;
      phaseCurrentL_3 : USInt;
      reserve_34818 : USInt;
      remainingMotorCoolingTime : UInt;
      reserve_34820 : USInt;
      asymmetry : USInt;
      motorTemperatureRise : UInt;
      reserve_34822 : UInt;
      reserve_34823 : UInt;
      reserve_34824 : UInt;
      outputFrequency : USInt;
      reserve_34825 : USInt;
      reserve_34826 : UInt;
      lineFrequency : USInt;
      reserve_34827 : USInt;
      "lineToLineVoltageL1-L2" : UInt;
      "lineToLineVoltageL2-L3" : UInt;
      "lineToLineVoltageL3-L1" : UInt;
      phaseCurrentL1RMS : DInt;
      phaseCurrentL2RMS : DInt;
      phaseCurrentL3RMS : DInt;
      reserve_34837 : UInt;
      reserve_34838 : USInt;
      switchingElementHeating : USInt;
      remainingSwitchingElementCoolingTime : UInt;
      remainingTimeForMotorOverloadProtection : UInt;
      activePower : DInt;
      reserve_34843 : UInt;
      "powerFactorL1-3" : USInt;
      reserve_34844 : USInt;
      reserve_34845 : UInt;
      reserve_34846 : UInt;
      reserve_34847 : UInt;
      remainingSwitchingFrequencyMonitoringTime : UInt;
      phaseCurrentAverage : USInt;
      reserve_34849 : USInt;
      reserve_34850 : UInt;
      phaseCurrentAverageRms : DInt;
      maximumPhaseCurrent : DInt;
      reserve_34855 : UInt;
      reserve_34856 : UInt;
      reserve_34857 : UInt;
      reserve_34858 : UInt;
      reserve_34859 : UInt;
      reserve_34860 : UInt;
   END_STRUCT;
END_TYPE

TYPE "typeStatisticData"
VERSION : 0.1
   STRUCT
      reserve_35840 : UInt;
      phaseMaximal : USInt;
      reserve_35841 : USInt;
      lastTripping : UInt;
      operatingHours : UDInt;
      numberOfMotorStartsRight : UDInt;
      numberOfMotorStartsLeft : UDInt;
      numberOfMotorOverloadTrips : UInt;
      reserve_35850 : UInt;
      maximumPhaseCurrent : DInt;
      lastTrippingCurrent : DInt;
      operatingHoursMotor : UDInt;
      operatingHoursMotorCurrent : UDInt;
      operatingHoursMotorCurrent1 : UDInt;
      operatingHoursMotorCurrent2 : UDInt;
      operatingHoursMotorCurrent3 : UDInt;
      reserve_35865 : UInt;
      numberOfSwitchingElementOverloadTrips : UInt;
      numberOfBypassOverloadTrips : UInt;
      reserve_35868 : UDInt;
      reserve_35870 : UInt;
      numberOfElectricalBrakingStops : UDInt;
      numberOfStartsOutput1 : UDInt;
      numberOfStartsOutput2 : UDInt;
      numberOfStartsOutput3 : UDInt;
      numberOfStartsOutput4 : UDInt;
      reserve_35881 : UDInt;
      reserve_35883 : UDInt;
      reserve_35885 : UDInt;
      reserve_35887 : UDInt;
      reserve_35889 : UDInt;
      reserve_35891 : UDInt;
      reserve_35893 : UDInt;
      reserve_35895 : UDInt;
      reserve_35897 : UDInt;
      activeEnergyImport : LReal;
      activeEnergyExport : LReal;
      lastRealStartingTime : UInt;
      reserve_35908 : UInt;
   END_STRUCT;
END_TYPE

TYPE "typeProcessImageOutput"
VERSION : 0.1
   STRUCT
      motorRight : Bool;
      motorLeft : Bool;
      reserve_33282 : Bool;
      reset : Bool;
      emergencyStart : Bool;
      selfTest : Bool;
      creepSpeed : Bool;
      reserve_33287 : Bool;
      output1 : Bool;
      output2 : Bool;
      parameterSetBit0 : Bool;
      parameterSetBit1 : Bool;
      reserve_33292 : Bool;
      reserve_33293 : Bool;
      reserve_33294 : Bool;
      disableQuickStop : Bool;
      output3 : Bool;
      reserve_33297 : Bool;
      reserve_33298 : Bool;
      pumpCleaning : Bool;
      reserve_33300 : Bool;
      reserve_33301 : Bool;
      reserve_33302 : Bool;
      reserve_33303 : Bool;
      manualOperationLocalInputControlled : Bool;
      useAlternativeStoppingMode : Bool;
      motorStandstill : Bool;
      reserve_33307 : Bool;
      reserve_33308 : Bool;
      reserve_33309 : Bool;
      reserve_33310 : Bool;
      reserve_33311 : Bool;
   END_STRUCT;
END_TYPE

TYPE "typeProcessImageInput"
VERSION : 0.1
   STRUCT
      ready : Bool;
      motorOn : Bool;
      groupError : Bool;
      groupWarning : Bool;
      input1 : Bool;
      input2 : Bool;
      input3 : Bool;
      input4 : Bool;
      motorCurrentLactBit0 : Bool;
      motorCurrentLactBit1 : Bool;
      motorCurrentLactBit2 : Bool;
      motorCurrentLactBit3 : Bool;
      motorCurrentLactBit4 : Bool;
      motorCurrentLactBit5 : Bool;
      manualOperationLocal : Bool;
      rampOperation : Bool;
      motorRight : Bool;
      motorLeft : Bool;
      reserve_32786 : Bool;
      reserve_32787 : Bool;
      startModeActive : Bool;
      operationBypassActive : Bool;
      stopModeActive : Bool;
      testOperationActive : Bool;
      thermalMotorModelOverload : Bool;
      temperatureSensorOverload : Bool;
      switchingElementOverload : Bool;
      coolingTimeActive : Bool;
      deviceError : Bool;
      automaticParameterizationActive : Bool;
      NewExParameterValuesDetected : Bool;
      reserve_32799 : Bool;
      measuredValue1 : Real;
      measuredValue2 : Real;
      measuredValue3 : Real;
   END_STRUCT;
END_TYPE

TYPE "typeModbusTcpCommunicationParameters"
VERSION : 0.1
   STRUCT
      reserve_41216 : UInt;
      reserve_41217 : UInt;
      accessMonitoringTime : UDInt;
      reserve_41220 : UDInt;
      reserve_41222 : UDInt;
      reserve_41224 : UDInt;
      reserve_41226 : UDInt;
      reserve_41228 : UDInt;
      ipAddress : Array[1..4] of Byte;
      subnetMask : Array[1..4] of Byte;
      routerAddress : Array[1..4] of Byte;
      macAddress : Byte;
      reserve_41236 : USInt;
      reserve_41237 : UInt;
      reserve_41238 : UInt;
   END_STRUCT;
END_TYPE

TYPE "typeMaximumPointer"
VERSION : 0.1
   STRUCT
      reserve_36864 : UInt;
      minimumPhaseCurrentL1 : USInt;
      minimumPhaseCurrentL2 : USInt;
      minimumPhaseCurrentL3 : USInt;
      reserve_36866 : USInt;
      maximumPhaseCurrentL1 : USInt;
      maximumPhaseCurrentL2 : USInt;
      maximumPhaseCurrentL3 : USInt;
      reserve_36868 : USInt;
      maximumTriggerCurrent : UInt;
      numberOfMotorOverloadTrips : UInt;
      maximumTriggerCurrent_1 : DInt;
      minimumPhaseCurrentL1RMS : DInt;
      minimumPhaseCurrentL2RMS : DInt;
      minimumPhaseCurrentL3RMS : DInt;
      maximumPhaseCurrentL1RMS : DInt;
      maximumPhaseCurrentL2RMS : DInt;
      maximumPhaseCurrentL3RMS : DInt;
      "lineToLineVoltageL1-L2Min" : UInt;
      "lineToLineVoltageL2-L3Min" : UInt;
      "lineToLineVoltageL3-L1Min" : UInt;
      "lineToLineVoltageL1-L2Max" : UInt;
      "lineToLineVoltageL2-L3Max" : UInt;
      "lineToLineVoltageL3-L1Max" : UInt;
      reserve_36891 : UInt;
      reserve_36892 : UInt;
      reserve_36893 : USInt;
      maximumSwitchingElementHeating : USInt;
      minimumLineFrequency : USInt;
      maximumLineFrequency : USInt;
      operatingHoursMotorCurrent : UDInt;
      operatingHoursMotorCurrent_1 : UDInt;
      operatingHoursMotorCurrent_2 : UDInt;
      operatingHoursMotorCurrent_3 : UDInt;
      operatingHoursDevice : UDInt;
      reserve_36905 : UInt;
      reserve_36906 : UInt;
      startingCurrentMaxRms : DInt;
      startingCurrentL1MaxRms : DInt;
      startingCurrentL2MaxRms : DInt;
      startingCurrentL3MaxRms : DInt;
      "numberOfStartsWithExt.Bypass" : UInt;
      reserve_36916 : UInt;
      reserve_36917 : UInt;
      reserve_36918 : UInt;
      reserve_36919 : UInt;
      reserve_36920 : UInt;
      reserve_36921 : UInt;
   END_STRUCT;
END_TYPE

TYPE "typeParameters"
VERSION : 0.1
   STRUCT
      reserve_37888 : UInt;
      automaticParameterization : Byte;
      reserve_37889 : Byte;
      presetStartingTime : UInt;
      control : UDInt;
      serviceFactor : Byte;
      reserve_37893 : USInt;
      ratedTorque : UInt;
      ratedOperatingSpeed : UInt;
      motorConnectionType : Byte;
      reserve_37896 : USInt;
      startingMode0 : Bool;
      startingMode1 : Bool;
      startingMode2 : Bool;
      startingMode3 : Bool;
      "reserve_37897.4" : Bool;
      "reserve_37897.5" : Bool;
      "reserve_37897.6" : Bool;
      "reserve_37897.7" : Bool;
      reserve_37897 : USInt;
      startVoltage : USInt;
      reserve_37898 : USInt;
      currentLimitingValue : UInt;
      startingTorque : USInt;
      reserve_37900 : USInt;
      limitingTorque : USInt;
      reserve_37901 : USInt;
      rampUpTime : UInt;
      maximumStartingTime : UInt;
      breakawayTime : USInt;
      reserve_37904 : USInt;
      breakawayVoltage : USInt;
      reserve_37905 : USInt;
      motorHeatingPower : USInt;
      reserve_37906 : USInt;
      stoppingMode0 : Bool;
      stoppingMode1 : Bool;
      stoppingMode2 : Bool;
      stoppingMode3 : Bool;
      "reserve_37907.4" : Bool;
      "reserve_37907.5" : Bool;
      "reserve_37907.6" : Bool;
      "reserve_37907.7" : Bool;
      reserve_37907 : USInt;
      stoppingTime : UInt;
      stoppingTorque : USInt;
      reserve_37909 : USInt;
      dynamicBrakingTorque : USInt;
      reserve_37910 : USInt;
      brakingTorqueDc : USInt;
      reserve_37911 : USInt;
      alternativeStoppingMode : Byte;
      reserve_37912 : USInt;
      alternativeStoppingTime : UInt;
      alternativeStoppingTorque : USInt;
      reserve_37914 : USInt;
      alternativeDynamicBrakingTorque : USInt;
      reserve_37915 : USInt;
      alternativeDcBrakingTorque : USInt;
      reserve_37916 : USInt;
      trippingClass : Byte;
      reserve_37917 : USInt;
      remainingTimeForTrippingWarningLimit : UInt;
      motorHeatingWarningLimit : USInt;
      reserve_37919 : USInt;
      responseToOverloadThermalMotorModel : Byte;
      reserve_37920 : USInt;
      recoveryTime : USInt;
      reserve_37921 : USInt;
      temperatureSensor0 : Bool;
      temperatureSensor1 : Bool;
      temperatureSensor2 : Bool;
      temperatureSensor3 : Bool;
      "reserve_37922.4" : Bool;
      "reserve_37922.5" : Bool;
      "reserve_37922.6" : Bool;
      "reserve_37922.7" : Bool;
      reserve_37922 : USInt;
      responseToOverloadTemperatureSensor : Bool;
      responseToOverloadTemperatureSensor1 : Bool;
      "reserve_37923.2" : Bool;
      "reserve_37923.3" : Bool;
      "reserve_37923.4" : Bool;
      "reserve_37923.5" : Bool;
      "reserve_37923.6" : Bool;
      "reserve_37923.7" : Bool;
      reserve_37923 : USInt;
      creepSpeedFactorRight : USInt;
      reserve_37924 : USInt;
      creepSpeedTorqueRight : USInt;
      reserve_37925 : USInt;
      creepSpeedFactorLeft : USInt;
      reserve_37926 : USInt;
      creepSpeedTorqueLeft : USInt;
      reserve_37927 : USInt;
      currentUpperLimitError : UInt;
      currentUpperLimitMaintenanceDemanded : UInt;
      currentLowerLimitError : USInt;
      reserve_37930 : USInt;
      currentLowerLimitMaintenanceDemanded : USInt;
      reserve_37931 : USInt;
      activePowerReferenceValue : UDInt;
      activePowerUpperLimitError : UInt;
      activePowerUpperLimitMaintenanceDemanded : UInt;
      activePowerLowerLimitError : USInt;
      reserve_37936 : USInt;
      activePowerLowerLimitMaintenanceDemanded : USInt;
      reserve_37937 : USInt;
      startingTimeUpperLimitMaintenanceDemanded : UInt;
      startingTimeLowerLimitMaintenanceDemanded : USInt;
      reserve_37939 : USInt;
      asymmetryLimitWarning : Byte;
      reserve_37940 : USInt;
      asymmetryLimitError : Byte;
      reserve_37941 : USInt;
      groundFaultLimitWarning : USInt;
      reserve_37942 : USInt;
      groundFaultLimitError : USInt;
      reserve_37943 : USInt;
      emergencyStart : Byte;
      reserve_37944 : USInt;
      reserve_37945 : UInt;
      input1Action : USInt;
      reserve_37946 : USInt;
      input2Action : USInt;
      reserve_37947 : USInt;
      input3Action : USInt;
      reserve_37948 : USInt;
      input4Action : USInt;
      reserve_37949 : USInt;
      output1Action : USInt;
      reserve_37950 : USInt;
      output1OnDelayTime : UInt;
      output1OffDelayTime : UInt;
      output2Action : USInt;
      reserve_37953 : USInt;
      output2OndelayTime : UInt;
      output2OffDelayTime : UInt;
      output4Action : USInt;
      reserve_37956 : USInt;
      output4OnDelayTime : UInt;
      output4OffDelayTime : UInt;
      analogOutputSignalType : USInt;
      reserve_37959 : USInt;
      analogOutputMeasuredValue : UInt;
      analogOutputRangeStartValue : UDInt;
      analogOutputRangeEndValue : UDInt;
      exApplication : Byte;
      reserve_37965 : USInt;
      responseToCpuMasterStop : Byte;
      reserve_37966 : USInt;
      substituteValueMotorRight : Bool;
      substituteValueMotorLeft : Bool;
      "reserve_37967.2" : Bool;
      substituteValueReset : Bool;
      substituteValueEmergencyStart : Bool;
      "reserve_37967.5" : Bool;
      substituteValueCreepSpeed : Bool;
      "reserve_37967.7" : Bool;
      substituteValueOutput1 : Bool;
      substituteValueOutput2 : Bool;
      substituteValueParameterSetBit0 : Bool;
      substituteValueParameterSetBit1 : Bool;
      "reserve_37967.12" : Bool;
      "reserve_37967.13" : Bool;
      "reserve_37967.14" : Bool;
      substituteValueDisableQuickStop : Bool;
      substituteValueOutput3 : Bool;
      "reserve_37968.1" : Bool;
      "reserve_37968.2" : Bool;
      substituteValuePumpCleaning : Bool;
      "reserve_37968.4" : Bool;
      "reserve_37968.5" : Bool;
      "reserve_37968.6" : Bool;
      "reserve_37968.7" : Bool;
      substituteValueManualOperationLocalInputControlled : Bool;
      substituteValueUseAlternativeStoppingMode : Bool;
      substituteValueMotorStandstill : Bool;
      "reserve_37968.11" : Bool;
      "reserve_37968.12" : Bool;
      "reserve_37968.13" : Bool;
      "reserve_37968.14" : Bool;
      "reserve_37968.15" : Bool;
      reserve_37969 : UInt;
      responseToOverloadSwitchingElement : Byte;
      reserve_37970 : USInt;
      responseToFaultyMainPower : Byte;
      reserve_37971 : USInt;
      responseToPresetUnequalActualConfigurationOfHmi : Byte;
      reserve_37972 : USInt;
      pumpCleaningMode : Byte;
      pumpCleaningStartStopParameters : Byte;
      pumpCleaningTime : USInt;
      pumpCleaningCycles : USInt;
      currentLimitingValueMaximum : UInt;
      reserve_37976 : UInt;
      reserve_37977 : UInt;
      reserve_37978 : UInt;
      reserve_37979 : UInt;
      measuredValue1 : UInt;
      measuredValue2 : UInt;
      measuredValue3 : UInt;
   END_STRUCT;
END_TYPE

TYPE "typeStatus"
VERSION : 0.1
   STRUCT
      error : Bool;
      status : Word;
      done : Bool;
      busy : Bool;
   END_STRUCT;
END_TYPE

TYPE "typeModbusRtuCommunicationParameters"
VERSION : 0.1
   STRUCT
      reserve_41472 : UDInt;
      accessMonitoringTime : UDInt;
      silentIntervalTime : UInt;
      reserve_41477 : UInt;
      baudRate : USInt;
      portConfiguration : USInt;
      stationAddress : USInt;
      reserve_41479 : USInt;
      detectedBaudRate : USInt;
      detectedPortConfiguration : USInt;
      reserve_41481 : UInt;
      reserve_41482 : UInt;
   END_STRUCT;
END_TYPE

TYPE "SoftStarterCOMM"
VERSION : 0.1
   STRUCT
      statusEstablishConnection : "typeStatus";
      requestReadProcessImageInput : Bool;
      requestReadProcessImageOutput : Bool;
      requestReadSoftStarterDiagnostics : Bool;
      requestReadMeasuredValues : Bool;
      requestReadStatisticData : Bool;
      requestReadMaximumPointer : Bool;
      requestReadParameters : Bool;
      requestWriteParameters : Bool;
      requestWriteProcessImageOutput : Bool;
      requestStartParameters : Bool;
      requestStopParameters : Bool;
      startingModeParameters : Int;
      stoppingModeParameters : Int;
      requestTemperatureSensorParameters : Bool;
      temperatureSensorParameters : Int;
      responseToOverloadTemperatureSensorParameters : Int;
      requestResponseToOverloadParameters : Bool;
      softStarterIdInput : Int;
      dataType : Struct
         dataSetProcessImageInput : "typeProcessImageInput";
         dataSetProcessImageOutput : "typeProcessImageOutput";
         dataSetSoftStarterDiagnostics : "typeSoftStarterDiagnostics";
         dataSetMeasuredValues : "typeMeasuredValues";
         dataSetStatisticData : "typeStatisticData";
         dataSetMaximumPointer : "typeMaximumPointer";
         dataSetParameters : "typeParameters";
      END_STRUCT;
   END_STRUCT;
END_TYPE

DATA_BLOCK "ANALOGAS"   // DB1
{ S7_Optimized_Access := 'TRUE' }
VERSION : 0.1
   VAR RETAIN
      "096PIT004" : Struct
         "CD MAX" : DInt := 27648;
         "CD MIN" : DInt := 0;
         "ING MAX" : Real := 232.0;
         "ING MIN" : Real := 0.0;
         HH : Real := 120.0;
         H : Real := 110.0;
         L : Real := 0.0;
         LL : Real := 1.5;
         ESCALIZADA : Real := 4.287905;
         PORCENTAJE : Real := 1.848235;
      END_STRUCT;
      "096PIT006" : Struct
         "CD MAX" : DInt := 27648;
         "CD MIN" : DInt := 0;
         "ING MAX" : Real := 232.0;
         "ING MIN" : Real := 0.0;
         HH : Real := 130.0;
         H : Real := 110.0;
         L : Real := 5.0;
         LL : Real := 0.0;
         ESCALIZADA : Real := 64.62905;
         PORCENTAJE : Real := 27.85735;
      END_STRUCT;
      "096PIT005" : Struct
         "CD MAX" : DInt := 27648;
         "CD MIN" : DInt := 0;
         "ING MAX" : Real := 232.0;
         "ING MIN" : Real := 0.0;
         HH : Real := 50.0;
         H : Real := 15.0;
         L : Real := 2.0;
         LL : Real := 1.5;
         ESCALIZADA : Real := 2.827836;
         PORCENTAJE : Real := 1.218895;
      END_STRUCT;
      "096PIT008" : Struct
         "CD MAX" : DInt := 27648;
         "CD MIN" : DInt := 0;
         "ING MAX" : Real := 232.0;
         "ING MIN" : Real := 0.0;
         HH : Real := 120.0;
         H : Real := 110.0;
         L : Real := 70.0;
         LL : Real := 1.0;
         ESCALIZADA : Real := 86.68113;
         PORCENTAJE : Real := 37.36256;
      END_STRUCT;
      "096PIT009" : Struct
         "CD MAX" : DInt := 27648;
         "CD MIN" : DInt := 0;
         "ING MAX" : Real := 232.0;
         "ING MIN" : Real := 0.0;
         HH : Real := 50.0;
         H : Real := 15.0;
         L : Real := 2.0;
         LL : Real := 1.5;
         ESCALIZADA : Real := 3.364872;
         PORCENTAJE : Real := 1.450376;
      END_STRUCT;
      "096PIT010" : Struct
         "CD MAX" : DInt := 27648;
         "CD MIN" : DInt := 0;
         "ING MAX" : Real := 232.0;
         "ING MIN" : Real := 0.0;
         HH : Real := 120.0;
         H : Real := 110.0;
         L : Real := 70.0;
         LL : Real := 20.0;
         ESCALIZADA : Real := 86.79021;
         PORCENTAJE : Real := 37.40958;
      END_STRUCT;
   END_VAR
BEGIN
END_DATA_BLOCK

